REGION Network 3: Reset counter for write modbus parameter
   RUNG wire#powerrail
      { S7_Templates := "SrcType := Int" } GT_Contact(in1 := "PCS1".iCountDoneW, in2 := 9)
      Move(in := 1, out1 => "PCS1".iCountDoneW)
   END_RUNG
   // the same network as SCL:
   IF "PCS1".iCountDoneW > 9 THEN "PCS1".iCountDoneW := 1; END_IF;
END_REGION

REGION Network 4: Counter for read modbus data value
   RUNG wire#powerrail
      N_Contact(operand := "MbPCS1_W".DONE, bit := "xPEP2")
      { S7_Templates := "SrcType := Int" } Add(in1 := "PCS1".iCountReadW, in2 := 1, out => "PCS1".iCountReadW)
   END_RUNG
   // the same network as SCL:
   #_w1 := NOT "MbPCS1_W".DONE AND "xPEP2";   // falling edge of "MbPCS1_W".DONE
   "xPEP2" := "MbPCS1_W".DONE;
   IF #_w1 THEN "PCS1".iCountReadW := "PCS1".iCountReadW + 1; END_IF;
END_REGION

REGION Network 5: Reset counter for read modbus data value
   RUNG wire#powerrail
      { S7_Templates := "SrcType := Int" } GT_Contact(in1 := "PCS1".iCountReadW, in2 := 9)
      Move(in := 1, out1 => "PCS1".iCountReadW)
   END_RUNG
   // the same network as SCL:
   IF "PCS1".iCountReadW > 9 THEN "PCS1".iCountReadW := 1; END_IF;
END_REGION

REGION Network 6: Set request data modbus
   RUNG wire#powerrail
      N_Contact(operand := "MbPCS1_W".DONE, bit := "xPEP3")
      S_Coil( "PCS1".xREQW )
   END_RUNG
   // the same network as SCL:
   #_w1 := NOT "MbPCS1_W".DONE AND "xPEP3";   // falling edge of "MbPCS1_W".DONE
   "xPEP3" := "MbPCS1_W".DONE;
   IF #_w1 THEN "PCS1".xREQW := TRUE; END_IF;
END_REGION

REGION Network 7: Reset request data modbus
   RUNG wire#powerrail
      P_Contact(operand := "MbPCS1_W".DONE, bit := "xPEP4")
      R_Coil( "PCS1".xREQW )
   END_RUNG
   // the same network as SCL:
   #_w1 := "MbPCS1_W".DONE AND NOT "xPEP4";   // rising edge of "MbPCS1_W".DONE
   "xPEP4" := "MbPCS1_W".DONE;
   IF #_w1 THEN "PCS1".xREQW := FALSE; END_IF;
END_REGION

REGION Network 9: Write W_Block1 parameter
   // wUserPswIns
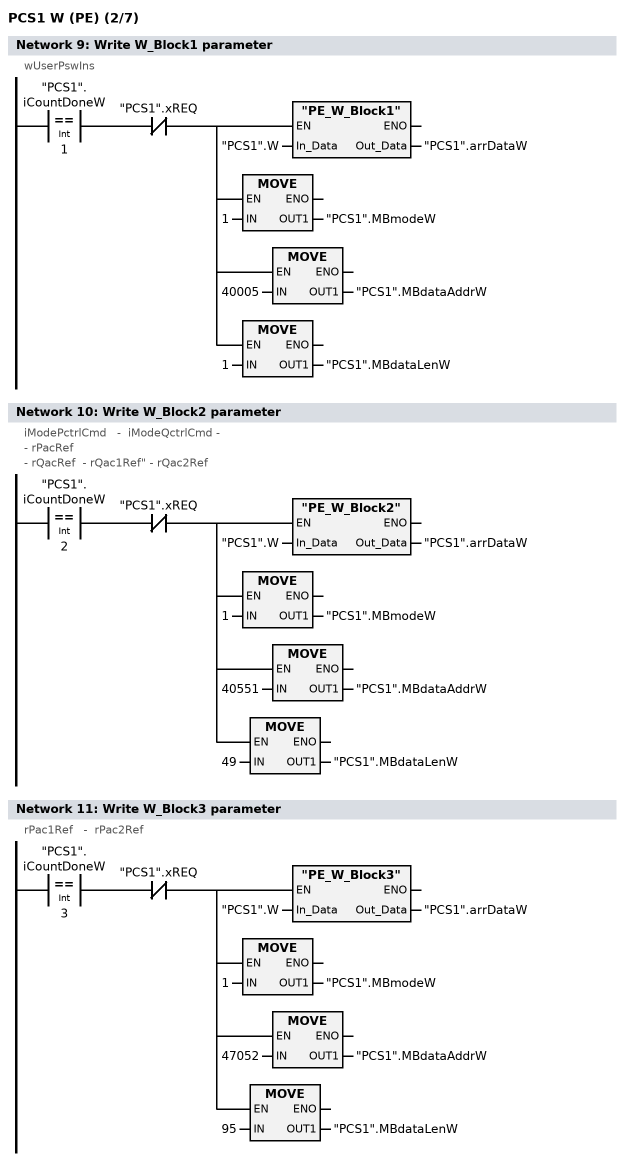
   RUNG wire#powerrail
      { S7_Templates := "SrcType := Int" } EQ_Contact(in1 := "PCS1".iCountDoneW, in2 := 1)
      I_Contact( "PCS1".xREQ )
      wire#w1
      "PE_W_Block1"(In_Data := "PCS1".W, Out_Data => "PCS1".arrDataW)
   END_RUNG
   RUNG wire#w1
      Move(in := 1, out1 => "PCS1".MBmodeW)
   END_RUNG
   RUNG wire#w1
      Move(in := 40005, out1 => "PCS1".MBdataAddrW)
   END_RUNG
   RUNG wire#w1
      Move(in := 1, out1 => "PCS1".MBdataLenW)
   END_RUNG
   // the same network as SCL:
   #_w1 := ("PCS1".iCountDoneW = 1) AND NOT "PCS1".xREQ;
   IF #_w1 THEN
       "PE_W_Block1"(In_Data := "PCS1".W, Out_Data => "PCS1".arrDataW);
       "PCS1".MBmodeW := 1;
       "PCS1".MBdataAddrW := 40005;
       "PCS1".MBdataLenW := 1;
   END_IF;
END_REGION

REGION Network 10: Write W_Block2 parameter
   // iModePctrlCmd   -  iModeQctrlCmd - 
   // - rPacRef 
   // - rQacRef  - rQac1Ref" - rQac2Ref
   RUNG wire#powerrail
      { S7_Templates := "SrcType := Int" } EQ_Contact(in1 := "PCS1".iCountDoneW, in2 := 2)
      I_Contact( "PCS1".xREQ )
      wire#w1
      "PE_W_Block2"(In_Data := "PCS1".W, Out_Data => "PCS1".arrDataW)
   END_RUNG
   RUNG wire#w1
      Move(in := 1, out1 => "PCS1".MBmodeW)
   END_RUNG
   RUNG wire#w1
      Move(in := 40551, out1 => "PCS1".MBdataAddrW)
   END_RUNG
   RUNG wire#w1
      Move(in := 49, out1 => "PCS1".MBdataLenW)
   END_RUNG
   // the same network as SCL:
   #_w1 := ("PCS1".iCountDoneW = 2) AND NOT "PCS1".xREQ;
   IF #_w1 THEN
       "PE_W_Block2"(In_Data := "PCS1".W, Out_Data => "PCS1".arrDataW);
       "PCS1".MBmodeW := 1;
       "PCS1".MBdataAddrW := 40551;
       "PCS1".MBdataLenW := 49;
   END_IF;
END_REGION

REGION Network 11: Write W_Block3 parameter
   // rPac1Ref   -  rPac2Ref
   RUNG wire#powerrail
      { S7_Templates := "SrcType := Int" } EQ_Contact(in1 := "PCS1".iCountDoneW, in2 := 3)
      I_Contact( "PCS1".xREQ )
      wire#w1
      "PE_W_Block3"(In_Data := "PCS1".W, Out_Data => "PCS1".arrDataW)
   END_RUNG
   RUNG wire#w1
      Move(in := 1, out1 => "PCS1".MBmodeW)
   END_RUNG
   RUNG wire#w1
      Move(in := 47052, out1 => "PCS1".MBdataAddrW)
   END_RUNG
   RUNG wire#w1
      Move(in := 95, out1 => "PCS1".MBdataLenW)
   END_RUNG
   // the same network as SCL:
   #_w1 := ("PCS1".iCountDoneW = 3) AND NOT "PCS1".xREQ;
   IF #_w1 THEN
       "PE_W_Block3"(In_Data := "PCS1".W, Out_Data => "PCS1".arrDataW);
       "PCS1".MBmodeW := 1;
       "PCS1".MBdataAddrW := 47052;
       "PCS1".MBdataLenW := 95;
   END_IF;
END_REGION

REGION Network 12: Write Command Start
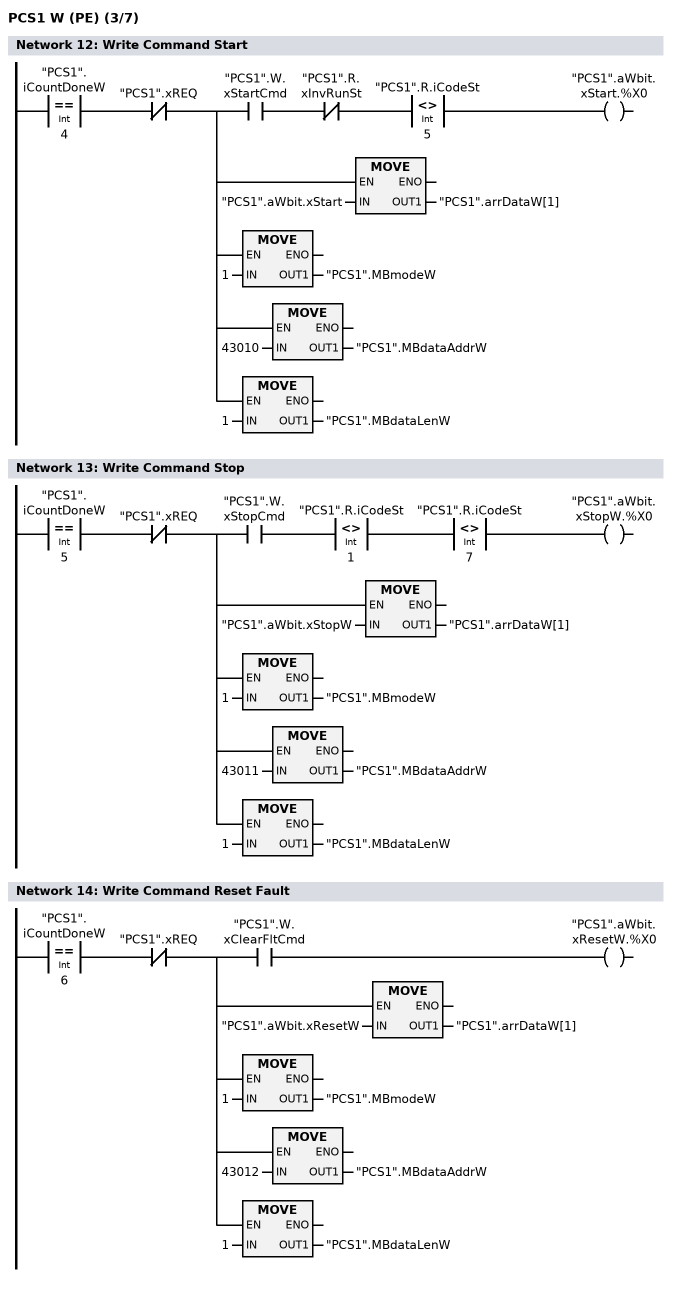
   RUNG wire#powerrail
      { S7_Templates := "SrcType := Int" } EQ_Contact(in1 := "PCS1".iCountDoneW, in2 := 4)
      I_Contact( "PCS1".xREQ )
      wire#w1
      Contact( "PCS1".W.xStartCmd )
      I_Contact( "PCS1".R.xInvRunSt )
      { S7_Templates := "SrcType := Int" } NE_Contact(in1 := "PCS1".R.iCodeSt, in2 := 5)
      Coil( "PCS1".aWbit.xStart.%X0 )
   END_RUNG
   RUNG wire#w1
      Move(in := "PCS1".aWbit.xStart, out1 => "PCS1".arrDataW[1])
   END_RUNG
   RUNG wire#w1
      Move(in := 1, out1 => "PCS1".MBmodeW)
   END_RUNG
   RUNG wire#w1
      Move(in := 43010, out1 => "PCS1".MBdataAddrW)
   END_RUNG
   RUNG wire#w1
      Move(in := 1, out1 => "PCS1".MBdataLenW)
   END_RUNG
   // the same network as SCL:
   #_w1 := ("PCS1".iCountDoneW = 4) AND NOT "PCS1".xREQ;
   "PCS1".aWbit.xStart.%X0 := #_w1 AND "PCS1".W.xStartCmd AND NOT "PCS1".R.xInvRunSt AND ("PCS1".R.iCodeSt <> 5);
   IF #_w1 THEN
       "PCS1".arrDataW[1] := "PCS1".aWbit.xStart;
       "PCS1".MBmodeW := 1;
       "PCS1".MBdataAddrW := 43010;
       "PCS1".MBdataLenW := 1;
   END_IF;
END_REGION

REGION Network 13: Write Command Stop
   RUNG wire#powerrail
      { S7_Templates := "SrcType := Int" } EQ_Contact(in1 := "PCS1".iCountDoneW, in2 := 5)
      I_Contact( "PCS1".xREQ )
      wire#w1
      Contact( "PCS1".W.xStopCmd )
      { S7_Templates := "SrcType := Int" } NE_Contact(in1 := "PCS1".R.iCodeSt, in2 := 1)
      { S7_Templates := "SrcType := Int" } NE_Contact(in1 := "PCS1".R.iCodeSt, in2 := 7)
      Coil( "PCS1".aWbit.xStopW.%X0 )
   END_RUNG
   RUNG wire#w1
      Move(in := "PCS1".aWbit.xStopW, out1 => "PCS1".arrDataW[1])
   END_RUNG
   RUNG wire#w1
      Move(in := 1, out1 => "PCS1".MBmodeW)
   END_RUNG
   RUNG wire#w1
      Move(in := 43011, out1 => "PCS1".MBdataAddrW)
   END_RUNG
   RUNG wire#w1
      Move(in := 1, out1 => "PCS1".MBdataLenW)
   END_RUNG
   // the same network as SCL:
   #_w1 := ("PCS1".iCountDoneW = 5) AND NOT "PCS1".xREQ;
   "PCS1".aWbit.xStopW.%X0 := #_w1 AND "PCS1".W.xStopCmd AND ("PCS1".R.iCodeSt <> 1) AND ("PCS1".R.iCodeSt <> 7);
   IF #_w1 THEN
       "PCS1".arrDataW[1] := "PCS1".aWbit.xStopW;
       "PCS1".MBmodeW := 1;
       "PCS1".MBdataAddrW := 43011;
       "PCS1".MBdataLenW := 1;
   END_IF;
END_REGION

REGION Network 14: Write Command Reset Fault
   RUNG wire#powerrail
      { S7_Templates := "SrcType := Int" } EQ_Contact(in1 := "PCS1".iCountDoneW, in2 := 6)
      I_Contact( "PCS1".xREQ )
      wire#w1
      Contact( "PCS1".W.xClearFltCmd )
      Coil( "PCS1".aWbit.xResetW.%X0 )
   END_RUNG
   RUNG wire#w1
      Move(in := "PCS1".aWbit.xResetW, out1 => "PCS1".arrDataW[1])
   END_RUNG
   RUNG wire#w1
      Move(in := 1, out1 => "PCS1".MBmodeW)
   END_RUNG
   RUNG wire#w1
      Move(in := 43012, out1 => "PCS1".MBdataAddrW)
   END_RUNG
   RUNG wire#w1
      Move(in := 1, out1 => "PCS1".MBdataLenW)
   END_RUNG
   // the same network as SCL:
   #_w1 := ("PCS1".iCountDoneW = 6) AND NOT "PCS1".xREQ;
   "PCS1".aWbit.xResetW.%X0 := #_w1 AND "PCS1".W.xClearFltCmd;
   IF #_w1 THEN
       "PCS1".arrDataW[1] := "PCS1".aWbit.xResetW;
       "PCS1".MBmodeW := 1;
       "PCS1".MBdataAddrW := 43012;
       "PCS1".MBdataLenW := 1;
   END_IF;
END_REGION

REGION Network 15: Write Command Enable Start/Stop
   // Con versione vecchia si usava solo questo registro per marcia ed arresto.
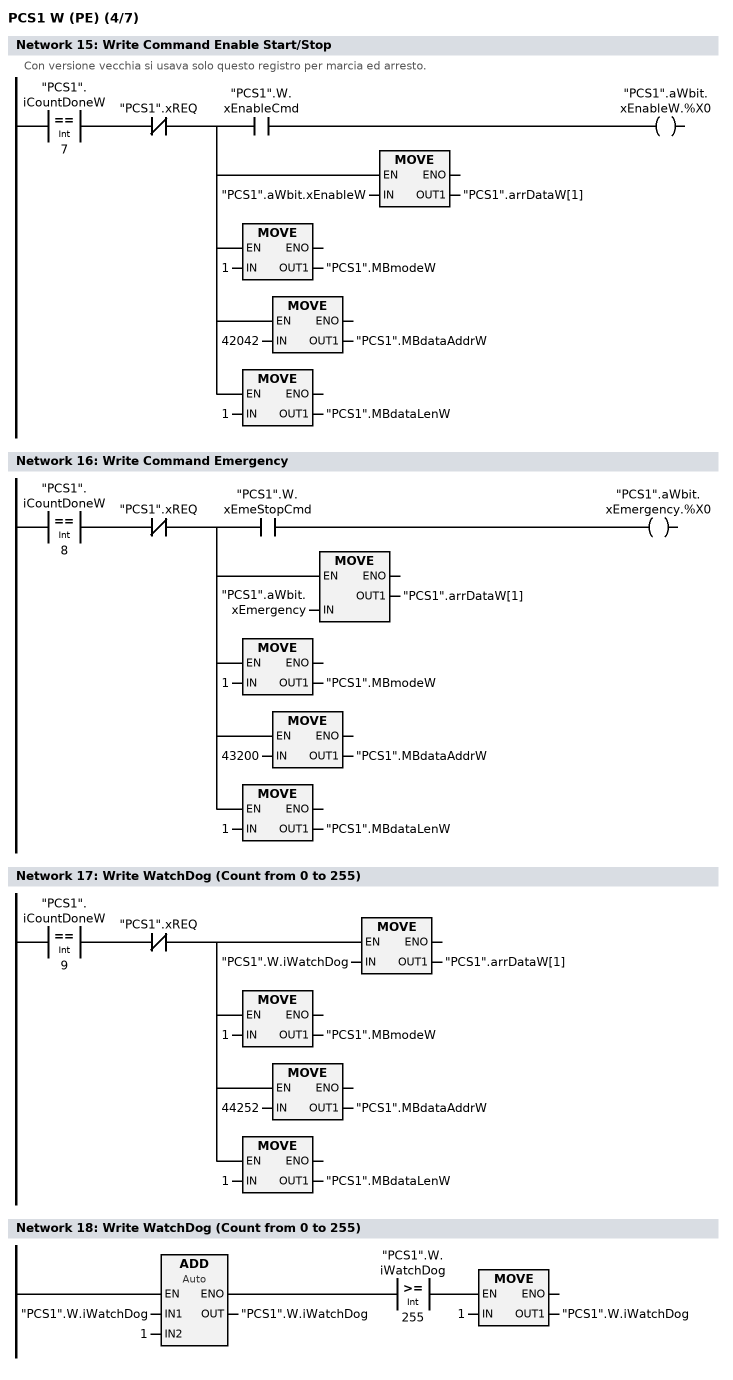
   RUNG wire#powerrail
      { S7_Templates := "SrcType := Int" } EQ_Contact(in1 := "PCS1".iCountDoneW, in2 := 7)
      I_Contact( "PCS1".xREQ )
      wire#w1
      Contact( "PCS1".W.xEnableCmd )
      Coil( "PCS1".aWbit.xEnableW.%X0 )
   END_RUNG
   RUNG wire#w1
      Move(in := "PCS1".aWbit.xEnableW, out1 => "PCS1".arrDataW[1])
   END_RUNG
   RUNG wire#w1
      Move(in := 1, out1 => "PCS1".MBmodeW)
   END_RUNG
   RUNG wire#w1
      Move(in := 42042, out1 => "PCS1".MBdataAddrW)
   END_RUNG
   RUNG wire#w1
      Move(in := 1, out1 => "PCS1".MBdataLenW)
   END_RUNG
   // the same network as SCL:
   #_w1 := ("PCS1".iCountDoneW = 7) AND NOT "PCS1".xREQ;
   "PCS1".aWbit.xEnableW.%X0 := #_w1 AND "PCS1".W.xEnableCmd;
   IF #_w1 THEN
       "PCS1".arrDataW[1] := "PCS1".aWbit.xEnableW;
       "PCS1".MBmodeW := 1;
       "PCS1".MBdataAddrW := 42042;
       "PCS1".MBdataLenW := 1;
   END_IF;
END_REGION

REGION Network 16: Write Command Emergency
   RUNG wire#powerrail
      { S7_Templates := "SrcType := Int" } EQ_Contact(in1 := "PCS1".iCountDoneW, in2 := 8)
      I_Contact( "PCS1".xREQ )
      wire#w1
      Contact( "PCS1".W.xEmeStopCmd )
      Coil( "PCS1".aWbit.xEmergency.%X0 )
   END_RUNG
   RUNG wire#w1
      Move(in := "PCS1".aWbit.xEmergency, out1 => "PCS1".arrDataW[1])
   END_RUNG
   RUNG wire#w1
      Move(in := 1, out1 => "PCS1".MBmodeW)
   END_RUNG
   RUNG wire#w1
      Move(in := 43200, out1 => "PCS1".MBdataAddrW)
   END_RUNG
   RUNG wire#w1
      Move(in := 1, out1 => "PCS1".MBdataLenW)
   END_RUNG
   // the same network as SCL:
   #_w1 := ("PCS1".iCountDoneW = 8) AND NOT "PCS1".xREQ;
   "PCS1".aWbit.xEmergency.%X0 := #_w1 AND "PCS1".W.xEmeStopCmd;
   IF #_w1 THEN
       "PCS1".arrDataW[1] := "PCS1".aWbit.xEmergency;
       "PCS1".MBmodeW := 1;
       "PCS1".MBdataAddrW := 43200;
       "PCS1".MBdataLenW := 1;
   END_IF;
END_REGION

REGION Network 17: Write WatchDog (Count from 0 to 255)
   RUNG wire#powerrail
      { S7_Templates := "SrcType := Int" } EQ_Contact(in1 := "PCS1".iCountDoneW, in2 := 9)
      I_Contact( "PCS1".xREQ )
      wire#w1
      Move(in := "PCS1".W.iWatchDog, out1 => "PCS1".arrDataW[1])
   END_RUNG
   RUNG wire#w1
      Move(in := 1, out1 => "PCS1".MBmodeW)
   END_RUNG
   RUNG wire#w1
      Move(in := 44252, out1 => "PCS1".MBdataAddrW)
   END_RUNG
   RUNG wire#w1
      Move(in := 1, out1 => "PCS1".MBdataLenW)
   END_RUNG
   // the same network as SCL:
   IF ("PCS1".iCountDoneW = 9) AND NOT "PCS1".xREQ THEN
       "PCS1".arrDataW[1] := "PCS1".W.iWatchDog;
       "PCS1".MBmodeW := 1;
       "PCS1".MBdataAddrW := 44252;
       "PCS1".MBdataLenW := 1;
   END_IF;
END_REGION

REGION Network 18: Write WatchDog (Count from 0 to 255)
   RUNG wire#powerrail
      Add(in1 := "PCS1".W.iWatchDog, in2 := 1, out => "PCS1".W.iWatchDog)
      { S7_Templates := "SrcType := Int" } GE_Contact(in1 := "PCS1".W.iWatchDog, in2 := 255)
      Move(in := 1, out1 => "PCS1".W.iWatchDog)
   END_RUNG
   // the same network as SCL:
   "PCS1".W.iWatchDog := "PCS1".W.iWatchDog + 1;
   IF "PCS1".W.iWatchDog >= 255 THEN "PCS1".W.iWatchDog := 1; END_IF;
END_REGION

REGION Network 20: 43010
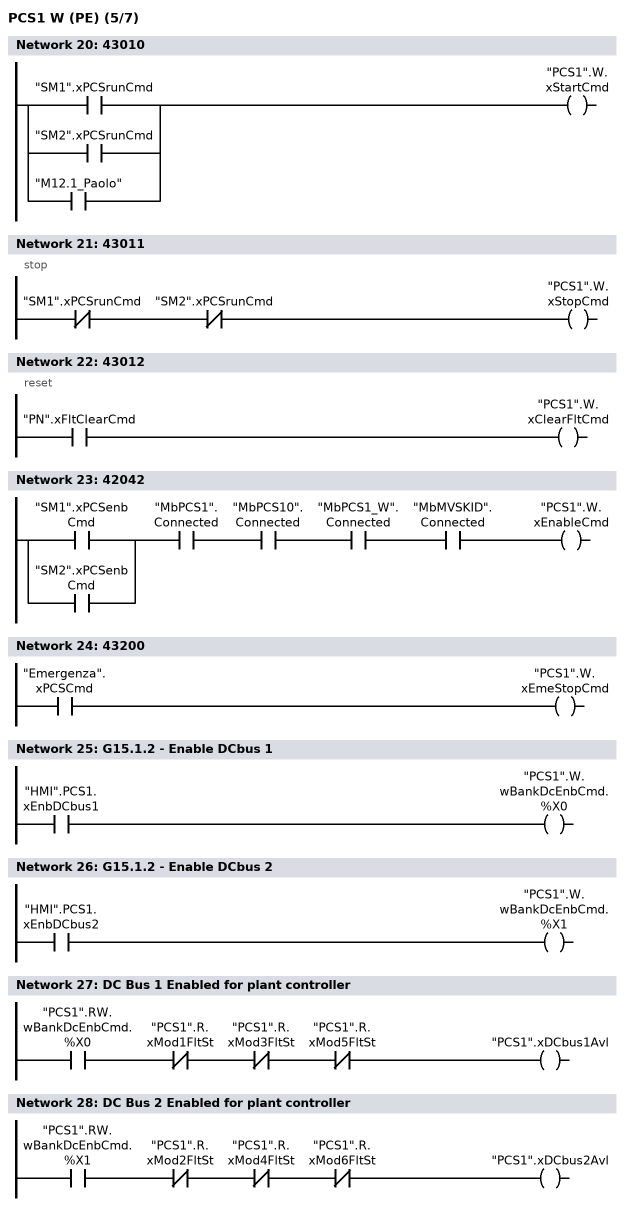
   RUNG wire#powerrail
      Contact( "SM1".xPCSrunCmd )
      wire#w1
      Coil( "PCS1".W.xStartCmd )
   END_RUNG
   RUNG wire#powerrail
      Contact( "SM2".xPCSrunCmd )
   END_RUNG wire#w1
   RUNG wire#powerrail
      Contact( "M12.1_Paolo" )
   END_RUNG wire#w1
   // the same network as SCL:
   "PCS1".W.xStartCmd := "SM1".xPCSrunCmd OR "SM2".xPCSrunCmd OR "M12.1_Paolo";
END_REGION

REGION Network 21: 43011
   // stop
   RUNG wire#powerrail
      I_Contact( "SM1".xPCSrunCmd )
      I_Contact( "SM2".xPCSrunCmd )
      Coil( "PCS1".W.xStopCmd )
   END_RUNG
   // the same network as SCL:
   "PCS1".W.xStopCmd := NOT "SM1".xPCSrunCmd AND NOT "SM2".xPCSrunCmd;
END_REGION

REGION Network 22: 43012
   // reset
   RUNG wire#powerrail
      Contact( "PN".xFltClearCmd )
      Coil( "PCS1".W.xClearFltCmd )
   END_RUNG
   // the same network as SCL:
   "PCS1".W.xClearFltCmd := "PN".xFltClearCmd;
END_REGION

REGION Network 23: 42042
   RUNG wire#powerrail
      Contact( "SM1".xPCSenbCmd )
      wire#w1
      Contact( "MbPCS1".Connected )
      Contact( "MbPCS10".Connected )
      Contact( "MbPCS1_W".Connected )
      Contact( "MbMVSKID".Connected )
      Coil( "PCS1".W.xEnableCmd )
   END_RUNG
   RUNG wire#powerrail
      Contact( "SM2".xPCSenbCmd )
   END_RUNG wire#w1
   // the same network as SCL:
   "PCS1".W.xEnableCmd := ("SM1".xPCSenbCmd OR "SM2".xPCSenbCmd) AND "MbPCS1".Connected AND "MbPCS10".Connected AND "MbPCS1_W".Connected AND "MbMVSKID".Connected;
END_REGION

REGION Network 24: 43200
   RUNG wire#powerrail
      Contact( "Emergenza".xPCSCmd )
      Coil( "PCS1".W.xEmeStopCmd )
   END_RUNG
   // the same network as SCL:
   "PCS1".W.xEmeStopCmd := "Emergenza".xPCSCmd;
END_REGION

REGION Network 25: G15.1.2 - Enable DCbus 1
   RUNG wire#powerrail
      Contact( "HMI".PCS1.xEnbDCbus1 )
      Coil( "PCS1".W.wBankDcEnbCmd.%X0 )
   END_RUNG
   // the same network as SCL:
   "PCS1".W.wBankDcEnbCmd.%X0 := "HMI".PCS1.xEnbDCbus1;
END_REGION

REGION Network 26: G15.1.2 - Enable DCbus 2
   RUNG wire#powerrail
      Contact( "HMI".PCS1.xEnbDCbus2 )
      Coil( "PCS1".W.wBankDcEnbCmd.%X1 )
   END_RUNG
   // the same network as SCL:
   "PCS1".W.wBankDcEnbCmd.%X1 := "HMI".PCS1.xEnbDCbus2;
END_REGION

REGION Network 27: DC Bus 1 Enabled for plant controller
   RUNG wire#powerrail
      Contact( "PCS1".RW.wBankDcEnbCmd.%X0 )
      I_Contact( "PCS1".R.xMod1FltSt )
      I_Contact( "PCS1".R.xMod3FltSt )
      I_Contact( "PCS1".R.xMod5FltSt )
      Coil( "PCS1".xDCbus1Avl )
   END_RUNG
   // the same network as SCL:
   "PCS1".xDCbus1Avl := "PCS1".RW.wBankDcEnbCmd.%X0 AND NOT "PCS1".R.xMod1FltSt AND NOT "PCS1".R.xMod3FltSt AND NOT "PCS1".R.xMod5FltSt;
END_REGION

REGION Network 28: DC Bus 2 Enabled for plant controller
   RUNG wire#powerrail
      Contact( "PCS1".RW.wBankDcEnbCmd.%X1 )
      I_Contact( "PCS1".R.xMod2FltSt )
      I_Contact( "PCS1".R.xMod4FltSt )
      I_Contact( "PCS1".R.xMod6FltSt )
      Coil( "PCS1".xDCbus2Avl )
   END_RUNG
   // the same network as SCL:
   "PCS1".xDCbus2Avl := "PCS1".RW.wBankDcEnbCmd.%X1 AND NOT "PCS1".R.xMod2FltSt AND NOT "PCS1".R.xMod4FltSt AND NOT "PCS1".R.xMod6FltSt;
END_REGION

REGION Network 30: Active Power local reference for PE with 2 DC Bus
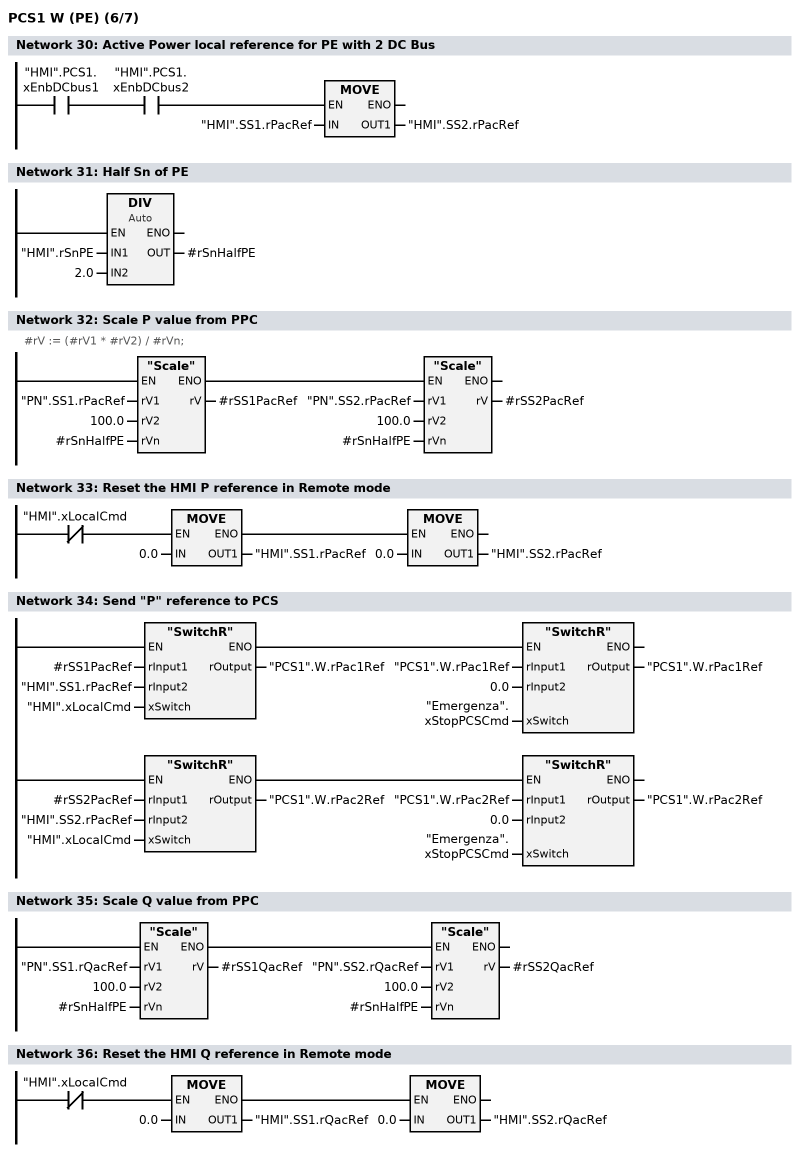
   RUNG wire#powerrail
      Contact( "HMI".PCS1.xEnbDCbus1 )
      Contact( "HMI".PCS1.xEnbDCbus2 )
      Move(in := "HMI".SS1.rPacRef, out1 => "HMI".SS2.rPacRef)
   END_RUNG
   // the same network as SCL:
   IF "HMI".PCS1.xEnbDCbus1 AND "HMI".PCS1.xEnbDCbus2 THEN "HMI".SS2.rPacRef := "HMI".SS1.rPacRef; END_IF;
END_REGION

REGION Network 31: Half Sn of PE
   RUNG wire#powerrail
      Div(in1 := "HMI".rSnPE, in2 := 2.0, out => #rSnHalfPE)
   END_RUNG
   // the same network as SCL:
   #rSnHalfPE := "HMI".rSnPE / 2.0;
END_REGION

REGION Network 32: Scale P value from PPC
   // #rV := (#rV1 * #rV2) / #rVn;
   RUNG wire#powerrail
      "Scale"(rV1 := "PN".SS1.rPacRef, rV2 := 100.0, rVn := #rSnHalfPE, rV => #rSS1PacRef)
      "Scale"(rV1 := "PN".SS2.rPacRef, rV2 := 100.0, rVn := #rSnHalfPE, rV => #rSS2PacRef)
   END_RUNG
   // the same network as SCL:
   "Scale"(rV1 := "PN".SS1.rPacRef, rV2 := 100.0, rVn := #rSnHalfPE, rV => #rSS1PacRef, ENO => #_w1);
   IF #_w1 THEN "Scale"(rV1 := "PN".SS2.rPacRef, rV2 := 100.0, rVn := #rSnHalfPE, rV => #rSS2PacRef); END_IF;
END_REGION

REGION Network 33: Reset the HMI P reference in Remote mode
   RUNG wire#powerrail
      I_Contact( "HMI".xLocalCmd )
      Move(in := 0.0, out1 => "HMI".SS1.rPacRef)
      Move(in := 0.0, out1 => "HMI".SS2.rPacRef)
   END_RUNG
   // the same network as SCL:
   IF NOT "HMI".xLocalCmd THEN
       "HMI".SS1.rPacRef := 0.0;
       "HMI".SS2.rPacRef := 0.0;
   END_IF;
END_REGION

REGION Network 34: Send "P" reference to PCS
   RUNG wire#powerrail
      "SwitchR"(rInput1 := #rSS1PacRef, rInput2 := "HMI".SS1.rPacRef, xSwitch := "HMI".xLocalCmd, rOutput => "PCS1".W.rPac1Ref)
      "SwitchR"(rInput1 := "PCS1".W.rPac1Ref, rInput2 := 0.0, xSwitch := "Emergenza".xStopPCSCmd, rOutput => "PCS1".W.rPac1Ref)
   END_RUNG
   RUNG wire#powerrail
      "SwitchR"(rInput1 := #rSS2PacRef, rInput2 := "HMI".SS2.rPacRef, xSwitch := "HMI".xLocalCmd, rOutput => "PCS1".W.rPac2Ref)
      "SwitchR"(rInput1 := "PCS1".W.rPac2Ref, rInput2 := 0.0, xSwitch := "Emergenza".xStopPCSCmd, rOutput => "PCS1".W.rPac2Ref)
   END_RUNG
   // the same network as SCL:
   "SwitchR"(rInput1 := #rSS1PacRef,
             rInput2 := "HMI".SS1.rPacRef,
             xSwitch := "HMI".xLocalCmd,
             rOutput => "PCS1".W.rPac1Ref,
             ENO => #_w1);
   IF #_w1 THEN
       "SwitchR"(rInput1 := "PCS1".W.rPac1Ref,
                 rInput2 := 0.0,
                 xSwitch := "Emergenza".xStopPCSCmd,
                 rOutput => "PCS1".W.rPac1Ref);
   END_IF;
   "SwitchR"(rInput1 := #rSS2PacRef,
             rInput2 := "HMI".SS2.rPacRef,
             xSwitch := "HMI".xLocalCmd,
             rOutput => "PCS1".W.rPac2Ref,
             ENO => #_w2);
   IF #_w2 THEN
       "SwitchR"(rInput1 := "PCS1".W.rPac2Ref,
                 rInput2 := 0.0,
                 xSwitch := "Emergenza".xStopPCSCmd,
                 rOutput => "PCS1".W.rPac2Ref);
   END_IF;
END_REGION

REGION Network 35: Scale Q value from PPC
   RUNG wire#powerrail
      "Scale"(rV1 := "PN".SS1.rQacRef, rV2 := 100.0, rVn := #rSnHalfPE, rV => #rSS1QacRef)
      "Scale"(rV1 := "PN".SS2.rQacRef, rV2 := 100.0, rVn := #rSnHalfPE, rV => #rSS2QacRef)
   END_RUNG
   // the same network as SCL:
   "Scale"(rV1 := "PN".SS1.rQacRef, rV2 := 100.0, rVn := #rSnHalfPE, rV => #rSS1QacRef, ENO => #_w1);
   IF #_w1 THEN "Scale"(rV1 := "PN".SS2.rQacRef, rV2 := 100.0, rVn := #rSnHalfPE, rV => #rSS2QacRef); END_IF;
END_REGION

REGION Network 36: Reset the HMI Q reference in Remote mode
   RUNG wire#powerrail
      I_Contact( "HMI".xLocalCmd )
      Move(in := 0.0, out1 => "HMI".SS1.rQacRef)
      Move(in := 0.0, out1 => "HMI".SS2.rQacRef)
   END_RUNG
   // the same network as SCL:
   IF NOT "HMI".xLocalCmd THEN
       "HMI".SS1.rQacRef := 0.0;
       "HMI".SS2.rQacRef := 0.0;
   END_IF;
END_REGION

REGION Network 37: Send "Q" reference to PCS
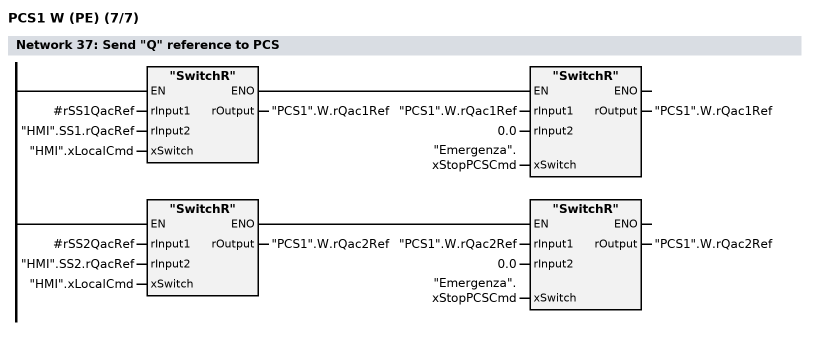
   RUNG wire#powerrail
      "SwitchR"(rInput1 := #rSS1QacRef, rInput2 := "HMI".SS1.rQacRef, xSwitch := "HMI".xLocalCmd, rOutput => "PCS1".W.rQac1Ref)
      "SwitchR"(rInput1 := "PCS1".W.rQac1Ref, rInput2 := 0.0, xSwitch := "Emergenza".xStopPCSCmd, rOutput => "PCS1".W.rQac1Ref)
   END_RUNG
   RUNG wire#powerrail
      "SwitchR"(rInput1 := #rSS2QacRef, rInput2 := "HMI".SS2.rQacRef, xSwitch := "HMI".xLocalCmd, rOutput => "PCS1".W.rQac2Ref)
      "SwitchR"(rInput1 := "PCS1".W.rQac2Ref, rInput2 := 0.0, xSwitch := "Emergenza".xStopPCSCmd, rOutput => "PCS1".W.rQac2Ref)
   END_RUNG
   // the same network as SCL:
   "SwitchR"(rInput1 := #rSS1QacRef,
             rInput2 := "HMI".SS1.rQacRef,
             xSwitch := "HMI".xLocalCmd,
             rOutput => "PCS1".W.rQac1Ref,
             ENO => #_w1);
   IF #_w1 THEN
       "SwitchR"(rInput1 := "PCS1".W.rQac1Ref,
                 rInput2 := 0.0,
                 xSwitch := "Emergenza".xStopPCSCmd,
                 rOutput => "PCS1".W.rQac1Ref);
   END_IF;
   "SwitchR"(rInput1 := #rSS2QacRef,
             rInput2 := "HMI".SS2.rQacRef,
             xSwitch := "HMI".xLocalCmd,
             rOutput => "PCS1".W.rQac2Ref,
             ENO => #_w2);
   IF #_w2 THEN
       "SwitchR"(rInput1 := "PCS1".W.rQac2Ref,
                 rInput2 := 0.0,
                 xSwitch := "Emergenza".xStopPCSCmd,
                 rOutput => "PCS1".W.rQac2Ref);
   END_IF;
END_REGION
END_FUNCTION

FUNCTION "PE_W_Block1" : Void
{ S7_Optimized_Access := 'TRUE' }
VERSION : 0.1
   VAR_INPUT 
      In_Data : "W_PE";   // pcs
   END_VAR

   VAR_OUTPUT 
      Out_Data : Array[1..125] of Word;
   END_VAR


BEGIN
	REGION
	    // 2022/01/24
	END_REGION
	
	REGION
	    
	    #Out_Data[1] := #In_Data."wUserPswIns";
	    
	END_REGION
END_FUNCTION

FUNCTION "PE_W_Block2" : Void
{ S7_Optimized_Access := 'TRUE' }
VERSION : 0.1
   VAR_INPUT 
      In_Data : "W_PE";   // udt. Samsung Data rack 1
   END_VAR

   VAR_OUTPUT 
      Out_Data : Array[1..125] of Word;
   END_VAR


BEGIN
	REGION
	    // 2022/01/24
	END_REGION
	
	REGION
	    
	    #Out_Data[1]    := INT_TO_WORD(#In_Data."iModePctrlCmd");
	    #Out_Data[2]    := INT_TO_WORD(#In_Data."iModeQctrlCmd");
	    #Out_Data[3]    := INT_TO_WORD(REAL_TO_INT((#In_Data."rPacRef")*100.0));
	    #Out_Data[8]    := INT_TO_WORD(REAL_TO_INT((#In_Data."rQacRef") * 100.0));
	    #Out_Data[48]   := INT_TO_WORD(REAL_TO_INT((#In_Data."rQac1Ref") * 100.0));
	    #Out_Data[49]   := INT_TO_WORD(REAL_TO_INT((#In_Data."rQac2Ref") * 100.0));
	    
	END_REGION
END_FUNCTION

FUNCTION "PE_W_Block3" : Void
{ S7_Optimized_Access := 'TRUE' }
VERSION : 0.1
   VAR_INPUT 
      In_Data : "W_PE";   // udt. Samsung Data rack 1
   END_VAR

   VAR_OUTPUT 
      Out_Data : Array[1..125] of Word;
   END_VAR


BEGIN
	REGION
	    // 2022/01/24
	END_REGION
	
	REGION
	    
	    #Out_Data[1]    := #In_Data."wBankDcEnbCmd";
	    #Out_Data[94]   := INT_TO_WORD(REAL_TO_INT((#In_Data."rPac1Ref")*100.0));
	    #Out_Data[95]   := INT_TO_WORD(REAL_TO_INT((#In_Data."rPac2Ref")*100.0));
	    
	END_REGION
END_FUNCTION

FUNCTION "Scale" : Void
{ S7_Optimized_Access := 'TRUE' }
VERSION : 0.1
   VAR_INPUT 
      rV1 : Real;
      rV2 : Real;
      rVn : Real;
   END_VAR

   VAR_OUTPUT 
      rV : Real;
   END_VAR


BEGIN
	
	#rV := (#rV1 * #rV2) / #rVn;
	
END_FUNCTION

FUNCTION "SwitchR" : Void
{ S7_Optimized_Access := 'TRUE' }
VERSION : 0.1
   VAR_INPUT 
      rInput1 : Real;
      rInput2 : Real;
      xSwitch : Bool;
   END_VAR

   VAR_OUTPUT 
      rOutput : Real;
   END_VAR

   VAR_TEMP 
      rOutTemp : Real;
   END_VAR


BEGIN
	IF #xSwitch THEN
	    #rOutTemp := #rInput2;
	ELSE
	    #rOutTemp := #rInput1;
	END_IF;
	
	#rOutput := #rOutTemp;
END_FUNCTION

FUNCTION "PN Com Read" : Void   // FC11, LAD
TITLE = ProfiNet Data Core <-> PEMS
{ S7_Optimized_Access := 'TRUE' }
VERSION : 0.1
// stored: AutoNumber false, IsIECCheckEnabled false, SetENOAutomatically false, UDAEnableTagReadback false
BEGIN

REGION Network 1: Read & Write Data From PEMS
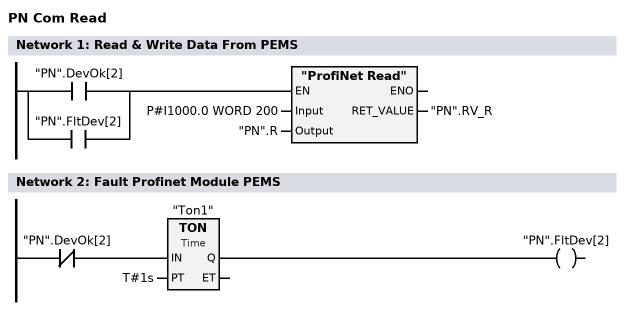
   RUNG wire#powerrail
      Contact( "PN".DevOk[2] )
      wire#w1
      "ProfiNet Read"(Input := P#I1000.0 WORD 200, Output := "PN".R, RET_VALUE => "PN".RV_R)
   END_RUNG
   RUNG wire#powerrail
      Contact( "PN".FltDev[2] )
   END_RUNG wire#w1
   // the same network as SCL:
   IF "PN".DevOk[2] OR "PN".FltDev[2] THEN
       "ProfiNet Read"(Input := P#I1000.0 WORD 200, Output := "PN".R, RET_VALUE => "PN".RV_R);
   END_IF;
END_REGION

REGION Network 2: Fault Profinet Module PEMS
   RUNG wire#powerrail
      I_Contact( "PN".DevOk[2] )
      { S7_Templates := "time_type := Time" } "Ton1".TON(pt := T#1s, et =>)
      Coil( "PN".FltDev[2] )
   END_RUNG
   // the same network as SCL:
   "Ton1".TON(IN := NOT "PN".DevOk[2], PT := T#1s);
   "PN".FltDev[2] := "Ton1".Q;
END_REGION
END_FUNCTION

FUNCTION "ProfiNet Read" : Void
{ S7_Optimized_Access := 'TRUE' }
VERSION : 0.1
   VAR_INPUT 
      Input : Variant;
   END_VAR

   VAR_OUTPUT 
      RET_VALUE : Int;
   END_VAR

   VAR_IN_OUT 
      Output : "PN Read";
   END_VAR

   VAR_TEMP 
      arrInput : Array[1..200] of Word;
      "DWORD" : DWord;
   END_VAR


BEGIN
	
	#RET_VALUE := MOVE_BLK_VARIANT(SRC := #Input, COUNT := 200, SRC_INDEX := 0, DEST_INDEX := 0, DEST => #arrInput);
	
	#Output."x1.1" := #arrInput[1].%X0;
	#Output."x1.2" := #arrInput[1].%X1;
	#Output."x1.3" := #arrInput[1].%X2;
	#Output."x1.4" := #arrInput[1].%X3;
	#Output."x1.5" := #arrInput[1].%X4;
	#Output."x1.6" := #arrInput[1].%X5;
	#Output."x1.7" := #arrInput[1].%X6;
	#Output."x1.8" := #arrInput[1].%X7;
	
	#Output."x2.1" := #arrInput[1].%X8;
	#Output."x2.2" := #arrInput[1].%X9;
	#Output."x2.3" := #arrInput[1].%X10;
	#Output."x2.4" := #arrInput[1].%X11;
	#Output."x2.5" := #arrInput[1].%X12;
	#Output."x2.6" := #arrInput[1].%X13;
	#Output."x2.7" := #arrInput[1].%X14;
	#Output."x2.8" := #arrInput[1].%X15;
	
	#Output."x3.1" := #arrInput[2].%X0;
	#Output."x3.2" := #arrInput[2].%X1;
	#Output."x3.3" := #arrInput[2].%X2;
	#Output."x3.4" := #arrInput[2].%X3;
	#Output."x3.5" := #arrInput[2].%X4;
	#Output."x3.6" := #arrInput[2].%X5;
	#Output."x3.7" := #arrInput[2].%X6;
	#Output."x3.8" := #arrInput[2].%X7;
	
	#Output."x4.1" := #arrInput[2].%X8;
	#Output."x4.2" := #arrInput[2].%X9;
	#Output."x4.3" := #arrInput[2].%X10;
	#Output."x4.4" := #arrInput[2].%X11;
	#Output."x4.5" := #arrInput[2].%X12;
	#Output."x4.6" := #arrInput[2].%X13;
	#Output."x4.7" := #arrInput[2].%X14;
	#Output."x4.8" := #arrInput[2].%X15;
	
	#Output."x5.1" := #arrInput[3].%X0;
	#Output."x5.2" := #arrInput[3].%X1;
	#Output."x5.3" := #arrInput[3].%X2;
	#Output."x5.4" := #arrInput[3].%X3;
	#Output."x5.5" := #arrInput[3].%X4;
	#Output."x5.6" := #arrInput[3].%X5;
	#Output."x5.7" := #arrInput[3].%X6;
	#Output."x5.8" := #arrInput[3].%X7;
	
	#Output."x6.1" := #arrInput[3].%X8;
	#Output."x6.2" := #arrInput[3].%X9;
	#Output."x6.3" := #arrInput[3].%X10;
	#Output."x6.4" := #arrInput[3].%X11;
	#Output."x6.5" := #arrInput[3].%X12;
	#Output."x6.6" := #arrInput[3].%X13;
	#Output."x6.7" := #arrInput[3].%X14;
	#Output."x6.8" := #arrInput[3].%X15;
	
	#Output."x7.1" := #arrInput[4].%X0;
	#Output."x7.2" := #arrInput[4].%X1;
	#Output."x7.3" := #arrInput[4].%X2;
	#Output."x7.4" := #arrInput[4].%X3;
	#Output."x7.5" := #arrInput[4].%X4;
	#Output."x7.6" := #arrInput[4].%X5;
	#Output."x7.7" := #arrInput[4].%X6;
	#Output."x7.8" := #arrInput[4].%X7;
	
	#Output."x8.1" := #arrInput[4].%X8;
	#Output."x8.2" := #arrInput[4].%X9;
	#Output."x8.3" := #arrInput[4].%X10;
	#Output."x8.4" := #arrInput[4].%X11;
	#Output."x8.5" := #arrInput[4].%X12;
	#Output."x8.6" := #arrInput[4].%X13;
	#Output."x8.7" := #arrInput[4].%X14;
	#Output."x8.8" := #arrInput[4].%X15;
	
	#Output."x9.1" := #arrInput[5].%X0;
	#Output."x9.2" := #arrInput[5].%X1;
	#Output."x9.3" := #arrInput[5].%X2;
	#Output."x9.4" := #arrInput[5].%X3;
	#Output."x9.5" := #arrInput[5].%X4;
	#Output."x9.6" := #arrInput[5].%X5;
	#Output."x9.7" := #arrInput[5].%X6;
	#Output."x9.8" := #arrInput[5].%X7;
	
	#Output."x10.1" := #arrInput[5].%X8;
	#Output."x10.2" := #arrInput[5].%X9;
	#Output."x10.3" := #arrInput[5].%X10;
	#Output."x10.4" := #arrInput[5].%X11;
	#Output."x10.5" := #arrInput[5].%X12;
	#Output."x10.6" := #arrInput[5].%X13;
	#Output."x10.7" := #arrInput[5].%X14;
	#Output."x10.8" := #arrInput[5].%X15;
	
	#Output.i1 := WORD_TO_INT(#arrInput[6]);
	#Output.i2 := WORD_TO_INT(#arrInput[7]);
	#Output.i3 := WORD_TO_INT(#arrInput[8]);
	#Output.i4 := WORD_TO_INT(#arrInput[9]);
	#Output.i5 := WORD_TO_INT(#arrInput[10]);
	#Output.i6 := WORD_TO_INT(#arrInput[11]);
	#Output.i7 := WORD_TO_INT(#arrInput[12]);
	#Output.i8 := WORD_TO_INT(#arrInput[13]);
	#Output.i9 := WORD_TO_INT(#arrInput[14]);
	#Output.i10 := WORD_TO_INT(#arrInput[15]);
	#Output.i11 := WORD_TO_INT(#arrInput[16]);
	#Output.i12 := WORD_TO_INT(#arrInput[17]);
	#Output.i13 := WORD_TO_INT(#arrInput[18]);
	#Output.i14 := WORD_TO_INT(#arrInput[19]);
	#Output.i15 := WORD_TO_INT(#arrInput[20]);
	#Output.i16 := WORD_TO_INT(#arrInput[21]);
	#Output.i17 := WORD_TO_INT(#arrInput[22]);
	#Output.i18 := WORD_TO_INT(#arrInput[23]);
	#Output.i19 := WORD_TO_INT(#arrInput[24]);
	#Output.i20 := WORD_TO_INT(#arrInput[25]);
	#Output.i21 := WORD_TO_INT(#arrInput[26]);
	#Output.i22 := WORD_TO_INT(#arrInput[27]);
	#Output.i23 := WORD_TO_INT(#arrInput[28]);
	#Output.i24 := WORD_TO_INT(#arrInput[29]);
	#Output.i25 := WORD_TO_INT(#arrInput[30]);
	#Output.i26 := WORD_TO_INT(#arrInput[31]);
	#Output.i27 := WORD_TO_INT(#arrInput[32]);
	#Output.i28 := WORD_TO_INT(#arrInput[33]);
	#Output.i29 := WORD_TO_INT(#arrInput[34]);
	#Output.i30 := WORD_TO_INT(#arrInput[35]);
	#Output.i31 := WORD_TO_INT(#arrInput[36]);
	#Output.i32 := WORD_TO_INT(#arrInput[37]);
	#Output.i33 := WORD_TO_INT(#arrInput[38]);
	#Output.i34 := WORD_TO_INT(#arrInput[39]);
	#Output.i35 := WORD_TO_INT(#arrInput[40]);
	
	#DWORD.%W0 := #arrInput[41];
	#DWORD.%W1 := #arrInput[42];
	#Output.r1 := DWORD_TO_REAL(#DWORD);
	#DWORD.%W0 := #arrInput[43];
	#DWORD.%W1 := #arrInput[44];
	#Output.r2 := DWORD_TO_REAL(#DWORD);
	#DWORD.%W0 := #arrInput[45];
	#DWORD.%W1 := #arrInput[46];
	#Output.r3 := DWORD_TO_REAL(#DWORD);
	#DWORD.%W0 := #arrInput[47];
	#DWORD.%W1 := #arrInput[48];
	#Output.r4 := DWORD_TO_REAL(#DWORD);
	#DWORD.%W0 := #arrInput[49];
	#DWORD.%W1 := #arrInput[50];
	#Output.r5 := DWORD_TO_REAL(#DWORD);
	#DWORD.%W0 := #arrInput[51];
	#DWORD.%W1 := #arrInput[52];
	#Output.r6 := DWORD_TO_REAL(#DWORD);
	#DWORD.%W0 := #arrInput[53];
	#DWORD.%W1 := #arrInput[54];
	#Output.r7 := DWORD_TO_REAL(#DWORD);
	#DWORD.%W0 := #arrInput[55];
	#DWORD.%W1 := #arrInput[56];
	#Output.r8 := DWORD_TO_REAL(#DWORD);
	#DWORD.%W0 := #arrInput[57];
	#DWORD.%W1 := #arrInput[58];
	#Output.r9 := DWORD_TO_REAL(#DWORD);
	#DWORD.%W0 := #arrInput[59];
	#DWORD.%W1 := #arrInput[60];
	#Output.r10 := DWORD_TO_REAL(#DWORD);
	#DWORD.%W0 := #arrInput[61];
	#DWORD.%W1 := #arrInput[62];
	#Output.r11 := DWORD_TO_REAL(#DWORD);
	#DWORD.%W0 := #arrInput[63];
	#DWORD.%W1 := #arrInput[64];
	#Output.r12 := DWORD_TO_REAL(#DWORD);
	#DWORD.%W0 := #arrInput[65];
	#DWORD.%W1 := #arrInput[66];
	#Output.r13 := DWORD_TO_REAL(#DWORD);
	#DWORD.%W0 := #arrInput[67];
	#DWORD.%W1 := #arrInput[68];
	#Output.r14 := DWORD_TO_REAL(#DWORD);
	#DWORD.%W0 := #arrInput[69];
	#DWORD.%W1 := #arrInput[70];
	#Output.r15 := DWORD_TO_REAL(#DWORD);
	#DWORD.%W0 := #arrInput[71];
	#DWORD.%W1 := #arrInput[72];
	#Output.r16 := DWORD_TO_REAL(#DWORD);
	#DWORD.%W0 := #arrInput[73];
	#DWORD.%W1 := #arrInput[74];
	#Output.r17 := DWORD_TO_REAL(#DWORD);
	#DWORD.%W0 := #arrInput[75];
	#DWORD.%W1 := #arrInput[76];
	#Output.r18 := DWORD_TO_REAL(#DWORD);
	#DWORD.%W0 := #arrInput[77];
	#DWORD.%W1 := #arrInput[78];
	#Output.r19 := DWORD_TO_REAL(#DWORD);
	#DWORD.%W0 := #arrInput[79];
	#DWORD.%W1 := #arrInput[80];
	#Output.r20 := DWORD_TO_REAL(#DWORD);
	#DWORD.%W0 := #arrInput[81];
	#DWORD.%W1 := #arrInput[82];
	#Output.r21 := DWORD_TO_REAL(#DWORD);
	#DWORD.%W0 := #arrInput[83];
	#DWORD.%W1 := #arrInput[84];
	#Output.r22 := DWORD_TO_REAL(#DWORD);
	#DWORD.%W0 := #arrInput[85];
	#DWORD.%W1 := #arrInput[86];
	#Output.r23 := DWORD_TO_REAL(#DWORD);
	#DWORD.%W0 := #arrInput[87];
	#DWORD.%W1 := #arrInput[88];
	#Output.r24 := DWORD_TO_REAL(#DWORD);
	#DWORD.%W0 := #arrInput[89];
	#DWORD.%W1 := #arrInput[90];
	#Output.r25 := DWORD_TO_REAL(#DWORD);
	#DWORD.%W0 := #arrInput[91];
	#DWORD.%W1 := #arrInput[92];
	#Output.r26 := DWORD_TO_REAL(#DWORD);
	#DWORD.%W0 := #arrInput[93];
	#DWORD.%W1 := #arrInput[94];
	#Output.r27 := DWORD_TO_REAL(#DWORD);
	#DWORD.%W0 := #arrInput[95];
	#DWORD.%W1 := #arrInput[96];
	#Output.r28 := DWORD_TO_REAL(#DWORD);
	#DWORD.%W0 := #arrInput[97];
	#DWORD.%W1 := #arrInput[98];
	#Output.r29 := DWORD_TO_REAL(#DWORD);
	#DWORD.%W0 := #arrInput[99];
	#DWORD.%W1 := #arrInput[100];
	#Output.r30 := DWORD_TO_REAL(#DWORD);
	#DWORD.%W0 := #arrInput[101];
	#DWORD.%W1 := #arrInput[102];
	#Output.r31 := DWORD_TO_REAL(#DWORD);
	#DWORD.%W0 := #arrInput[103];
	#DWORD.%W1 := #arrInput[104];
	#Output.r32 := DWORD_TO_REAL(#DWORD);
	#DWORD.%W0 := #arrInput[105];
	#DWORD.%W1 := #arrInput[106];
	#Output.r33 := DWORD_TO_REAL(#DWORD);
	#DWORD.%W0 := #arrInput[107];
	#DWORD.%W1 := #arrInput[108];
	#Output.r34 := DWORD_TO_REAL(#DWORD);
	#DWORD.%W0 := #arrInput[109];
	#DWORD.%W1 := #arrInput[110];
	#Output.r35 := DWORD_TO_REAL(#DWORD);
	#DWORD.%W0 := #arrInput[111];
	#DWORD.%W1 := #arrInput[112];
	#Output.r36 := DWORD_TO_REAL(#DWORD);
	#DWORD.%W0 := #arrInput[113];
	#DWORD.%W1 := #arrInput[114];
	#Output.r37 := DWORD_TO_REAL(#DWORD);
	#DWORD.%W0 := #arrInput[115];
	#DWORD.%W1 := #arrInput[116];
	#Output.r38 := DWORD_TO_REAL(#DWORD);
	#DWORD.%W0 := #arrInput[117];
	#DWORD.%W1 := #arrInput[118];
	#Output.r39 := DWORD_TO_REAL(#DWORD);
	#DWORD.%W0 := #arrInput[119];
	#DWORD.%W1 := #arrInput[120];
	#Output.r40 := DWORD_TO_REAL(#DWORD);
	#DWORD.%W0 := #arrInput[121];
	#DWORD.%W1 := #arrInput[122];
	#Output.r41 := DWORD_TO_REAL(#DWORD);
	#DWORD.%W0 := #arrInput[123];
	#DWORD.%W1 := #arrInput[124];
	#Output.r42 := DWORD_TO_REAL(#DWORD);
	#DWORD.%W0 := #arrInput[125];
	#DWORD.%W1 := #arrInput[126];
	#Output.r43 := DWORD_TO_REAL(#DWORD);
	#DWORD.%W0 := #arrInput[127];
	#DWORD.%W1 := #arrInput[128];
	#Output.r44 := DWORD_TO_REAL(#DWORD);
	#DWORD.%W0 := #arrInput[129];
	#DWORD.%W1 := #arrInput[130];
	#Output.r45 := DWORD_TO_REAL(#DWORD);
	#DWORD.%W0 := #arrInput[131];
	#DWORD.%W1 := #arrInput[132];
	#Output.r46 := DWORD_TO_REAL(#DWORD);
	#DWORD.%W0 := #arrInput[133];
	#DWORD.%W1 := #arrInput[134];
	#Output.r47 := DWORD_TO_REAL(#DWORD);
	#DWORD.%W0 := #arrInput[135];
	#DWORD.%W1 := #arrInput[136];
	#Output.r48 := DWORD_TO_REAL(#DWORD);
	#DWORD.%W0 := #arrInput[137];
	#DWORD.%W1 := #arrInput[138];
	#Output.r49 := DWORD_TO_REAL(#DWORD);
	#DWORD.%W0 := #arrInput[139];
	#DWORD.%W1 := #arrInput[140];
	#Output.r50 := DWORD_TO_REAL(#DWORD);
	#DWORD.%W0 := #arrInput[141];
	#DWORD.%W1 := #arrInput[142];
	#Output.r51 := DWORD_TO_REAL(#DWORD);
	#DWORD.%W0 := #arrInput[143];
	#DWORD.%W1 := #arrInput[144];
	#Output.r52 := DWORD_TO_REAL(#DWORD);
	#DWORD.%W0 := #arrInput[145];
	#DWORD.%W1 := #arrInput[146];
	#Output.r53 := DWORD_TO_REAL(#DWORD);
	#DWORD.%W0 := #arrInput[147];
	#DWORD.%W1 := #arrInput[148];
	#Output.r54 := DWORD_TO_REAL(#DWORD);
	#DWORD.%W0 := #arrInput[149];
	#DWORD.%W1 := #arrInput[150];
	#Output.r55 := DWORD_TO_REAL(#DWORD);
	#DWORD.%W0 := #arrInput[151];
	#DWORD.%W1 := #arrInput[152];
	#Output.r56 := DWORD_TO_REAL(#DWORD);
	#DWORD.%W0 := #arrInput[153];
	#DWORD.%W1 := #arrInput[154];
	#Output.r57 := DWORD_TO_REAL(#DWORD);
	#DWORD.%W0 := #arrInput[155];
	#DWORD.%W1 := #arrInput[156];
	#Output.r58 := DWORD_TO_REAL(#DWORD);
	#DWORD.%W0 := #arrInput[157];
	#DWORD.%W1 := #arrInput[158];
	#Output.r59 := DWORD_TO_REAL(#DWORD);
	#DWORD.%W0 := #arrInput[159];
	#DWORD.%W1 := #arrInput[160];
	#Output.r60 := DWORD_TO_REAL(#DWORD);
	#DWORD.%W0 := #arrInput[161];
	#DWORD.%W1 := #arrInput[162];
	#Output.r61 := DWORD_TO_REAL(#DWORD);
	#DWORD.%W0 := #arrInput[163];
	#DWORD.%W1 := #arrInput[164];
	#Output.r62 := DWORD_TO_REAL(#DWORD);
	#DWORD.%W0 := #arrInput[165];
	#DWORD.%W1 := #arrInput[166];
	#Output.r63 := DWORD_TO_REAL(#DWORD);
	#DWORD.%W0 := #arrInput[167];
	#DWORD.%W1 := #arrInput[168];
	#Output.r64 := DWORD_TO_REAL(#DWORD);
	#DWORD.%W0 := #arrInput[169];
	#DWORD.%W1 := #arrInput[170];
	#Output.r65 := DWORD_TO_REAL(#DWORD);
	#DWORD.%W0 := #arrInput[171];
	#DWORD.%W1 := #arrInput[172];
	#Output.r66 := DWORD_TO_REAL(#DWORD);
	#DWORD.%W0 := #arrInput[173];
	#DWORD.%W1 := #arrInput[174];
	#Output.r67 := DWORD_TO_REAL(#DWORD);
	#DWORD.%W0 := #arrInput[175];
	#DWORD.%W1 := #arrInput[176];
	#Output.r68 := DWORD_TO_REAL(#DWORD);
	#DWORD.%W0 := #arrInput[177];
	#DWORD.%W1 := #arrInput[178];
	#Output.r69 := DWORD_TO_REAL(#DWORD);
	#DWORD.%W0 := #arrInput[179];
	#DWORD.%W1 := #arrInput[180];
	#Output.r70 := DWORD_TO_REAL(#DWORD);
	#DWORD.%W0 := #arrInput[181];
	#DWORD.%W1 := #arrInput[182];
	#Output.r71 := DWORD_TO_REAL(#DWORD);
	#DWORD.%W0 := #arrInput[183];
	#DWORD.%W1 := #arrInput[184];
	#Output.r72 := DWORD_TO_REAL(#DWORD);
	#DWORD.%W0 := #arrInput[185];
	#DWORD.%W1 := #arrInput[186];
	#Output.r73 := DWORD_TO_REAL(#DWORD);
	#DWORD.%W0 := #arrInput[187];
	#DWORD.%W1 := #arrInput[188];
	#Output.r74 := DWORD_TO_REAL(#DWORD);
	#DWORD.%W0 := #arrInput[189];
	#DWORD.%W1 := #arrInput[190];
	#Output.r75 := DWORD_TO_REAL(#DWORD);
	#DWORD.%W0 := #arrInput[191];
	#DWORD.%W1 := #arrInput[192];
	#Output.r76 := DWORD_TO_REAL(#DWORD);
	#DWORD.%W0 := #arrInput[193];
	#DWORD.%W1 := #arrInput[194];
	#Output.r77 := DWORD_TO_REAL(#DWORD);
	#DWORD.%W0 := #arrInput[195];
	#DWORD.%W1 := #arrInput[196];
	#Output.r78 := DWORD_TO_REAL(#DWORD);
	#DWORD.%W0 := #arrInput[197];
	#DWORD.%W1 := #arrInput[198];
	#Output.r79 := DWORD_TO_REAL(#DWORD);
	#DWORD.%W0 := #arrInput[199];
	#DWORD.%W1 := #arrInput[200];
	#Output.r80 := DWORD_TO_REAL(#DWORD);
	
END_FUNCTION

FUNCTION "PN Com Write" : Void   // FC12, LAD
TITLE = ProfiNet Data Core <-> PEMS
{ S7_Optimized_Access := 'TRUE' }
VERSION : 0.1
// stored: AutoNumber false, IsIECCheckEnabled false, SetENOAutomatically false, UDAEnableTagReadback false
BEGIN

REGION Network 1: Read & Write Data From PEMS
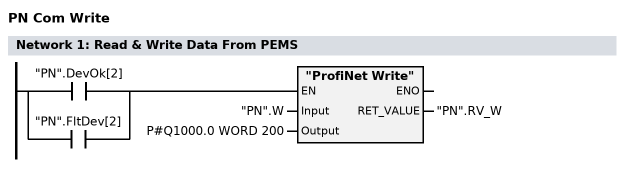
   RUNG wire#powerrail
      Contact( "PN".DevOk[2] )
      wire#w1
      "ProfiNet Write"(Input := "PN".W, Output := P#Q1000.0 WORD 200, RET_VALUE => "PN".RV_W)
   END_RUNG
   RUNG wire#powerrail
      Contact( "PN".FltDev[2] )
   END_RUNG wire#w1
   // the same network as SCL:
   IF "PN".DevOk[2] OR "PN".FltDev[2] THEN
       "ProfiNet Write"(Input := "PN".W, Output := P#Q1000.0 WORD 200, RET_VALUE => "PN".RV_W);
   END_IF;
END_REGION
END_FUNCTION

FUNCTION "ProfiNet Write" : Void
{ S7_Optimized_Access := 'TRUE' }
VERSION : 0.1
   VAR_INPUT 
      Input : "PN Write";
   END_VAR

   VAR_OUTPUT 
      RET_VALUE : Int;
   END_VAR

   VAR_IN_OUT 
      Output : Variant;
   END_VAR

   VAR_TEMP 
      arrOutput : Array[1..200] of Word;
      "DWORD" : DWord;
   END_VAR


BEGIN
	
	#arrOutput[1].%X0 := #Input."x1.1";
	#arrOutput[1].%X1 := #Input."x1.2";
	#arrOutput[1].%X2 := #Input."x1.3";
	#arrOutput[1].%X3 := #Input."x1.4";
	#arrOutput[1].%X4 := #Input."x1.5";
	#arrOutput[1].%X5 := #Input."x1.6";
	#arrOutput[1].%X6 := #Input."x1.7";
	#arrOutput[1].%X7 := #Input."x1.8";
	
	#arrOutput[1].%X8 := #Input."x2.1";
	#arrOutput[1].%X9 := #Input."x2.2";
	#arrOutput[1].%X10 := #Input."x2.3";
	#arrOutput[1].%X11 := #Input."x2.4";
	#arrOutput[1].%X12 := #Input."x2.5";
	#arrOutput[1].%X13 := #Input."x2.6";
	#arrOutput[1].%X14 := #Input."x2.7";
	#arrOutput[1].%X15 := #Input."x2.8";
	
	#arrOutput[2].%X0 := #Input."x3.1";
	#arrOutput[2].%X1 := #Input."x3.2";
	#arrOutput[2].%X2 := #Input."x3.3";
	#arrOutput[2].%X3 := #Input."x3.4";
	#arrOutput[2].%X4 := #Input."x3.5";
	#arrOutput[2].%X5 := #Input."x3.6";
	#arrOutput[2].%X6 := #Input."x3.7";
	#arrOutput[2].%X7 := #Input."x3.8";
	
	#arrOutput[2].%X8 := #Input."x4.1";
	#arrOutput[2].%X9 := #Input."x4.2";
	#arrOutput[2].%X10 := #Input."x4.3";
	#arrOutput[2].%X11 := #Input."x4.4";
	#arrOutput[2].%X12 := #Input."x4.5";
	#arrOutput[2].%X13 := #Input."x4.6";
	#arrOutput[2].%X14 := #Input."x4.7";
	#arrOutput[2].%X15 := #Input."x4.8";
	
	#arrOutput[3].%X0 := #Input."x5.1";
	#arrOutput[3].%X1 := #Input."x5.2";
	#arrOutput[3].%X2 := #Input."x5.3";
	#arrOutput[3].%X3 := #Input."x5.4";
	#arrOutput[3].%X4 := #Input."x5.5";
	#arrOutput[3].%X5 := #Input."x5.6";
	#arrOutput[3].%X6 := #Input."x5.7";
	#arrOutput[3].%X7 := #Input."x5.8";
	
	#arrOutput[3].%X8 := #Input."x6.1";
	#arrOutput[3].%X9 := #Input."x6.2";
	#arrOutput[3].%X10 := #Input."x6.3";
	#arrOutput[3].%X11 := #Input."x6.4";
	#arrOutput[3].%X12 := #Input."x6.5";
	#arrOutput[3].%X13 := #Input."x6.6";
	#arrOutput[3].%X14 := #Input."x6.7";
	#arrOutput[3].%X15 := #Input."x6.8";
	
	#arrOutput[4].%X0 := #Input."x7.1";
	#arrOutput[4].%X1 := #Input."x7.2";
	#arrOutput[4].%X2 := #Input."x7.3";
	#arrOutput[4].%X3 := #Input."x7.4";
	#arrOutput[4].%X4 := #Input."x7.5";
	#arrOutput[4].%X5 := #Input."x7.6";
	#arrOutput[4].%X6 := #Input."x7.7";
	#arrOutput[4].%X7 := #Input."x7.8";
	
	#arrOutput[4].%X8 := #Input."x8.1";
	#arrOutput[4].%X9 := #Input."x8.2";
	#arrOutput[4].%X10 := #Input."x8.3";
	#arrOutput[4].%X11 := #Input."x8.4";
	#arrOutput[4].%X12 := #Input."x8.5";
	#arrOutput[4].%X13 := #Input."x8.6";
	#arrOutput[4].%X14 := #Input."x8.7";
	#arrOutput[4].%X15 := #Input."x8.8";
	
	#arrOutput[5].%X0 := #Input."x9.1";
	#arrOutput[5].%X1 := #Input."x9.2";
	#arrOutput[5].%X2 := #Input."x9.3";
	#arrOutput[5].%X3 := #Input."x9.4";
	#arrOutput[5].%X4 := #Input."x9.5";
	#arrOutput[5].%X5 := #Input."x9.6";
	#arrOutput[5].%X6 := #Input."x9.7";
	#arrOutput[5].%X7 := #Input."x9.8";
	
	#arrOutput[5].%X8 := #Input."x10.1";
	#arrOutput[5].%X9 := #Input."x10.2";
	#arrOutput[5].%X10 := #Input."x10.3";
	#arrOutput[5].%X11 := #Input."x10.4";
	#arrOutput[5].%X12 := #Input."x10.5";
	#arrOutput[5].%X13 := #Input."x10.6";
	#arrOutput[5].%X14 := #Input."x10.7";
	#arrOutput[5].%X15 := #Input."x10.8";
	
	#arrOutput[6] := INT_TO_WORD(#Input.i1);
	#arrOutput[7] := INT_TO_WORD(#Input.i2);
	#arrOutput[8] := INT_TO_WORD(#Input.i3);
	#arrOutput[9] := INT_TO_WORD(#Input.i4);
	#arrOutput[10] := INT_TO_WORD(#Input.i5);
	#arrOutput[11] := INT_TO_WORD(#Input.i6);
	#arrOutput[12] := INT_TO_WORD(#Input.i7);
	#arrOutput[13] := INT_TO_WORD(#Input.i8);
	#arrOutput[14] := INT_TO_WORD(#Input.i9);
	#arrOutput[15] := INT_TO_WORD(#Input.i10);
	#arrOutput[16] := INT_TO_WORD(#Input.i11);
	#arrOutput[17] := INT_TO_WORD(#Input.i12);
	#arrOutput[18] := INT_TO_WORD(#Input.i13);
	#arrOutput[19] := INT_TO_WORD(#Input.i14);
	#arrOutput[20] := INT_TO_WORD(#Input.i15);
	#arrOutput[21] := INT_TO_WORD(#Input.i16);
	#arrOutput[22] := INT_TO_WORD(#Input.i17);
	#arrOutput[23] := INT_TO_WORD(#Input.i18);
	#arrOutput[24] := INT_TO_WORD(#Input.i19);
	#arrOutput[25] := INT_TO_WORD(#Input.i20);
	#arrOutput[26] := INT_TO_WORD(#Input.i21);
	#arrOutput[27] := INT_TO_WORD(#Input.i22);
	#arrOutput[28] := INT_TO_WORD(#Input.i23);
	#arrOutput[29] := INT_TO_WORD(#Input.i24);
	#arrOutput[30] := INT_TO_WORD(#Input.i25);
	#arrOutput[31] := INT_TO_WORD(#Input.i26);
	#arrOutput[32] := INT_TO_WORD(#Input.i27);
	#arrOutput[33] := INT_TO_WORD(#Input.i28);
	#arrOutput[34] := INT_TO_WORD(#Input.i29);
	#arrOutput[35] := INT_TO_WORD(#Input.i30);
	#arrOutput[36] := INT_TO_WORD(#Input.i31);
	#arrOutput[37] := INT_TO_WORD(#Input.i32);
	#arrOutput[38] := INT_TO_WORD(#Input.i33);
	#arrOutput[39] := INT_TO_WORD(#Input.i34);
	#arrOutput[40] := INT_TO_WORD(#Input.i35);
	
	#DWORD := REAL_TO_DWORD(#Input.r1);
	#arrOutput[41] := #DWORD.%W0;
	#arrOutput[42] := #DWORD.%W1;
	#DWORD := REAL_TO_DWORD(#Input.r2);
	#arrOutput[43] := #DWORD.%W0;
	#arrOutput[44] := #DWORD.%W1;
	#DWORD := REAL_TO_DWORD(#Input.r3);
	#arrOutput[45] := #DWORD.%W0;
	#arrOutput[46] := #DWORD.%W1;
	#DWORD := REAL_TO_DWORD(#Input.r4);
	#arrOutput[47] := #DWORD.%W0;
	#arrOutput[48] := #DWORD.%W1;
	#DWORD := REAL_TO_DWORD(#Input.r5);
	#arrOutput[49] := #DWORD.%W0;
	#arrOutput[50] := #DWORD.%W1;
	#DWORD := REAL_TO_DWORD(#Input.r6);
	#arrOutput[51] := #DWORD.%W0;
	#arrOutput[52] := #DWORD.%W1;
	#DWORD := REAL_TO_DWORD(#Input.r7);
	#arrOutput[53] := #DWORD.%W0;
	#arrOutput[54] := #DWORD.%W1;
	#DWORD := REAL_TO_DWORD(#Input.r8);
	#arrOutput[55] := #DWORD.%W0;
	#arrOutput[56] := #DWORD.%W1;
	#DWORD := REAL_TO_DWORD(#Input.r9);
	#arrOutput[57] := #DWORD.%W0;
	#arrOutput[58] := #DWORD.%W1;
	#DWORD := REAL_TO_DWORD(#Input.r10);
	#arrOutput[59] := #DWORD.%W0;
	#arrOutput[60] := #DWORD.%W1;
	#DWORD := REAL_TO_DWORD(#Input.r11);
	#arrOutput[61] := #DWORD.%W0;
	#arrOutput[62] := #DWORD.%W1;
	#DWORD := REAL_TO_DWORD(#Input.r12);
	#arrOutput[63] := #DWORD.%W0;
	#arrOutput[64] := #DWORD.%W1;
	#DWORD := REAL_TO_DWORD(#Input.r13);
	#arrOutput[65] := #DWORD.%W0;
	#arrOutput[66] := #DWORD.%W1;
	#DWORD := REAL_TO_DWORD(#Input.r14);
	#arrOutput[67] := #DWORD.%W0;
	#arrOutput[68] := #DWORD.%W1;
	#DWORD := REAL_TO_DWORD(#Input.r15);
	#arrOutput[69] := #DWORD.%W0;
	#arrOutput[70] := #DWORD.%W1;
	#DWORD := REAL_TO_DWORD(#Input.r16);
	#arrOutput[71] := #DWORD.%W0;
	#arrOutput[72] := #DWORD.%W1;
	#DWORD := REAL_TO_DWORD(#Input.r17);
	#arrOutput[73] := #DWORD.%W0;
	#arrOutput[74] := #DWORD.%W1;
	#DWORD := REAL_TO_DWORD(#Input.r18);
	#arrOutput[75] := #DWORD.%W0;
	#arrOutput[76] := #DWORD.%W1;
	#DWORD := REAL_TO_DWORD(#Input.r19);
	#arrOutput[77] := #DWORD.%W0;
	#arrOutput[78] := #DWORD.%W1;
	#DWORD := REAL_TO_DWORD(#Input.r20);
	#arrOutput[79] := #DWORD.%W0;
	#arrOutput[80] := #DWORD.%W1;
	#DWORD := REAL_TO_DWORD(#Input.r21);
	#arrOutput[81] := #DWORD.%W0;
	#arrOutput[82] := #DWORD.%W1;
	#DWORD := REAL_TO_DWORD(#Input.r22);
	#arrOutput[83] := #DWORD.%W0;
	#arrOutput[84] := #DWORD.%W1;
	#DWORD := REAL_TO_DWORD(#Input.r23);
	#arrOutput[85] := #DWORD.%W0;
	#arrOutput[86] := #DWORD.%W1;
	#DWORD := REAL_TO_DWORD(#Input.r24);
	#arrOutput[87] := #DWORD.%W0;
	#arrOutput[88] := #DWORD.%W1;
	#DWORD := REAL_TO_DWORD(#Input.r25);
	#arrOutput[89] := #DWORD.%W0;
	#arrOutput[90] := #DWORD.%W1;
	#DWORD := REAL_TO_DWORD(#Input.r26);
	#arrOutput[91] := #DWORD.%W0;
	#arrOutput[92] := #DWORD.%W1;
	#DWORD := REAL_TO_DWORD(#Input.r27);
	#arrOutput[93] := #DWORD.%W0;
	#arrOutput[94] := #DWORD.%W1;
	#DWORD := REAL_TO_DWORD(#Input.r28);
	#arrOutput[95] := #DWORD.%W0;
	#arrOutput[96] := #DWORD.%W1;
	#DWORD := REAL_TO_DWORD(#Input.r29);
	#arrOutput[97] := #DWORD.%W0;
	#arrOutput[98] := #DWORD.%W1;
	#DWORD := REAL_TO_DWORD(#Input.r30);
	#arrOutput[99] := #DWORD.%W0;
	#arrOutput[100] := #DWORD.%W1;
	#DWORD := REAL_TO_DWORD(#Input.r31);
	#arrOutput[101] := #DWORD.%W0;
	#arrOutput[102] := #DWORD.%W1;
	#DWORD := REAL_TO_DWORD(#Input.r32);
	#arrOutput[103] := #DWORD.%W0;
	#arrOutput[104] := #DWORD.%W1;
	#DWORD := REAL_TO_DWORD(#Input.r33);
	#arrOutput[105] := #DWORD.%W0;
	#arrOutput[106] := #DWORD.%W1;
	#DWORD := REAL_TO_DWORD(#Input.r34);
	#arrOutput[107] := #DWORD.%W0;
	#arrOutput[108] := #DWORD.%W1;
	#DWORD := REAL_TO_DWORD(#Input.r35);
	#arrOutput[109] := #DWORD.%W0;
	#arrOutput[110] := #DWORD.%W1;
	#DWORD := REAL_TO_DWORD(#Input.r36);
	#arrOutput[111] := #DWORD.%W0;
	#arrOutput[112] := #DWORD.%W1;
	#DWORD := REAL_TO_DWORD(#Input.r37);
	#arrOutput[113] := #DWORD.%W0;
	#arrOutput[114] := #DWORD.%W1;
	#DWORD := REAL_TO_DWORD(#Input.r38);
	#arrOutput[115] := #DWORD.%W0;
	#arrOutput[116] := #DWORD.%W1;
	#DWORD := REAL_TO_DWORD(#Input.r39);
	#arrOutput[117] := #DWORD.%W0;
	#arrOutput[118] := #DWORD.%W1;
	#DWORD := REAL_TO_DWORD(#Input.r40);
	#arrOutput[119] := #DWORD.%W0;
	#arrOutput[120] := #DWORD.%W1;
	#DWORD := REAL_TO_DWORD(#Input.r41);
	#arrOutput[121] := #DWORD.%W0;
	#arrOutput[122] := #DWORD.%W1;
	#DWORD := REAL_TO_DWORD(#Input.r42);
	#arrOutput[123] := #DWORD.%W0;
	#arrOutput[124] := #DWORD.%W1;
	#DWORD := REAL_TO_DWORD(#Input.r43);
	#arrOutput[125] := #DWORD.%W0;
	#arrOutput[126] := #DWORD.%W1;
	#DWORD := REAL_TO_DWORD(#Input.r44);
	#arrOutput[127] := #DWORD.%W0;
	#arrOutput[128] := #DWORD.%W1;
	#DWORD := REAL_TO_DWORD(#Input.r45);
	#arrOutput[129] := #DWORD.%W0;
	#arrOutput[130] := #DWORD.%W1;
	#DWORD := REAL_TO_DWORD(#Input.r46);
	#arrOutput[131] := #DWORD.%W0;
	#arrOutput[132] := #DWORD.%W1;
	#DWORD := REAL_TO_DWORD(#Input.r47);
	#arrOutput[133] := #DWORD.%W0;
	#arrOutput[134] := #DWORD.%W1;
	#DWORD := REAL_TO_DWORD(#Input.r48);
	#arrOutput[135] := #DWORD.%W0;
	#arrOutput[136] := #DWORD.%W1;
	#DWORD := REAL_TO_DWORD(#Input.r49);
	#arrOutput[137] := #DWORD.%W0;
	#arrOutput[138] := #DWORD.%W1;
	#DWORD := REAL_TO_DWORD(#Input.r50);
	#arrOutput[139] := #DWORD.%W0;
	#arrOutput[140] := #DWORD.%W1;
	#DWORD := REAL_TO_DWORD(#Input.r51);
	#arrOutput[141] := #DWORD.%W0;
	#arrOutput[142] := #DWORD.%W1;
	#DWORD := REAL_TO_DWORD(#Input.r52);
	#arrOutput[143] := #DWORD.%W0;
	#arrOutput[144] := #DWORD.%W1;
	#DWORD := REAL_TO_DWORD(#Input.r53);
	#arrOutput[145] := #DWORD.%W0;
	#arrOutput[146] := #DWORD.%W1;
	#DWORD := REAL_TO_DWORD(#Input.r54);
	#arrOutput[147] := #DWORD.%W0;
	#arrOutput[148] := #DWORD.%W1;
	#DWORD := REAL_TO_DWORD(#Input.r55);
	#arrOutput[149] := #DWORD.%W0;
	#arrOutput[150] := #DWORD.%W1;
	#DWORD := REAL_TO_DWORD(#Input.r56);
	#arrOutput[151] := #DWORD.%W0;
	#arrOutput[152] := #DWORD.%W1;
	#DWORD := REAL_TO_DWORD(#Input.r57);
	#arrOutput[153] := #DWORD.%W0;
	#arrOutput[154] := #DWORD.%W1;
	#DWORD := REAL_TO_DWORD(#Input.r58);
	#arrOutput[155] := #DWORD.%W0;
	#arrOutput[156] := #DWORD.%W1;
	#DWORD := REAL_TO_DWORD(#Input.r59);
	#arrOutput[157] := #DWORD.%W0;
	#arrOutput[158] := #DWORD.%W1;
	#DWORD := REAL_TO_DWORD(#Input.r60);
	#arrOutput[159] := #DWORD.%W0;
	#arrOutput[160] := #DWORD.%W1;
	#DWORD := REAL_TO_DWORD(#Input.r61);
	#arrOutput[161] := #DWORD.%W0;
	#arrOutput[162] := #DWORD.%W1;
	#DWORD := REAL_TO_DWORD(#Input.r62);
	#arrOutput[163] := #DWORD.%W0;
	#arrOutput[164] := #DWORD.%W1;
	#DWORD := REAL_TO_DWORD(#Input.r63);
	#arrOutput[165] := #DWORD.%W0;
	#arrOutput[166] := #DWORD.%W1;
	#DWORD := REAL_TO_DWORD(#Input.r64);
	#arrOutput[167] := #DWORD.%W0;
	#arrOutput[168] := #DWORD.%W1;
	#DWORD := REAL_TO_DWORD(#Input.r65);
	#arrOutput[169] := #DWORD.%W0;
	#arrOutput[170] := #DWORD.%W1;
	#DWORD := REAL_TO_DWORD(#Input.r66);
	#arrOutput[171] := #DWORD.%W0;
	#arrOutput[172] := #DWORD.%W1;
	#DWORD := REAL_TO_DWORD(#Input.r67);
	#arrOutput[173] := #DWORD.%W0;
	#arrOutput[174] := #DWORD.%W1;
	#DWORD := REAL_TO_DWORD(#Input.r68);
	#arrOutput[175] := #DWORD.%W0;
	#arrOutput[176] := #DWORD.%W1;
	#DWORD := REAL_TO_DWORD(#Input.r69);
	#arrOutput[177] := #DWORD.%W0;
	#arrOutput[178] := #DWORD.%W1;
	#DWORD := REAL_TO_DWORD(#Input.r70);
	#arrOutput[179] := #DWORD.%W0;
	#arrOutput[180] := #DWORD.%W1;
	#DWORD := REAL_TO_DWORD(#Input.r71);
	#arrOutput[181] := #DWORD.%W0;
	#arrOutput[182] := #DWORD.%W1;
	#DWORD := REAL_TO_DWORD(#Input.r72);
	#arrOutput[183] := #DWORD.%W0;
	#arrOutput[184] := #DWORD.%W1;
	#DWORD := REAL_TO_DWORD(#Input.r73);
	#arrOutput[185] := #DWORD.%W0;
	#arrOutput[186] := #DWORD.%W1;
	#DWORD := REAL_TO_DWORD(#Input.r74);
	#arrOutput[187] := #DWORD.%W0;
	#arrOutput[188] := #DWORD.%W1;
	#DWORD := REAL_TO_DWORD(#Input.r75);
	#arrOutput[189] := #DWORD.%W0;
	#arrOutput[190] := #DWORD.%W1;
	#DWORD := REAL_TO_DWORD(#Input.r76);
	#arrOutput[191] := #DWORD.%W0;
	#arrOutput[192] := #DWORD.%W1;
	#DWORD := REAL_TO_DWORD(#Input.r77);
	#arrOutput[193] := #DWORD.%W0;
	#arrOutput[194] := #DWORD.%W1;
	#DWORD := REAL_TO_DWORD(#Input.r78);
	#arrOutput[195] := #DWORD.%W0;
	#arrOutput[196] := #DWORD.%W1;
	#DWORD := REAL_TO_DWORD(#Input.r79);
	#arrOutput[197] := #DWORD.%W0;
	#arrOutput[198] := #DWORD.%W1;
	#DWORD := REAL_TO_DWORD(#Input.r80);
	#arrOutput[199] := #DWORD.%W0;
	#arrOutput[200] := #DWORD.%W1;
	
	#RET_VALUE := MOVE_BLK_VARIANT(SRC := #arrOutput, COUNT := 200, SRC_INDEX := 0, DEST_INDEX := 0, DEST => #Output);
	
END_FUNCTION

FUNCTION_BLOCK "Main_Safety_RTG1"   // FB501, F_LAD
{ S7_Optimized_Access := 'TRUE' }
VERSION : 0.1
// stored: AutoNumber false, IsIECCheckEnabled false, UDAEnableTagReadback false
BEGIN

REGION Network 1: Receive data from Core - new
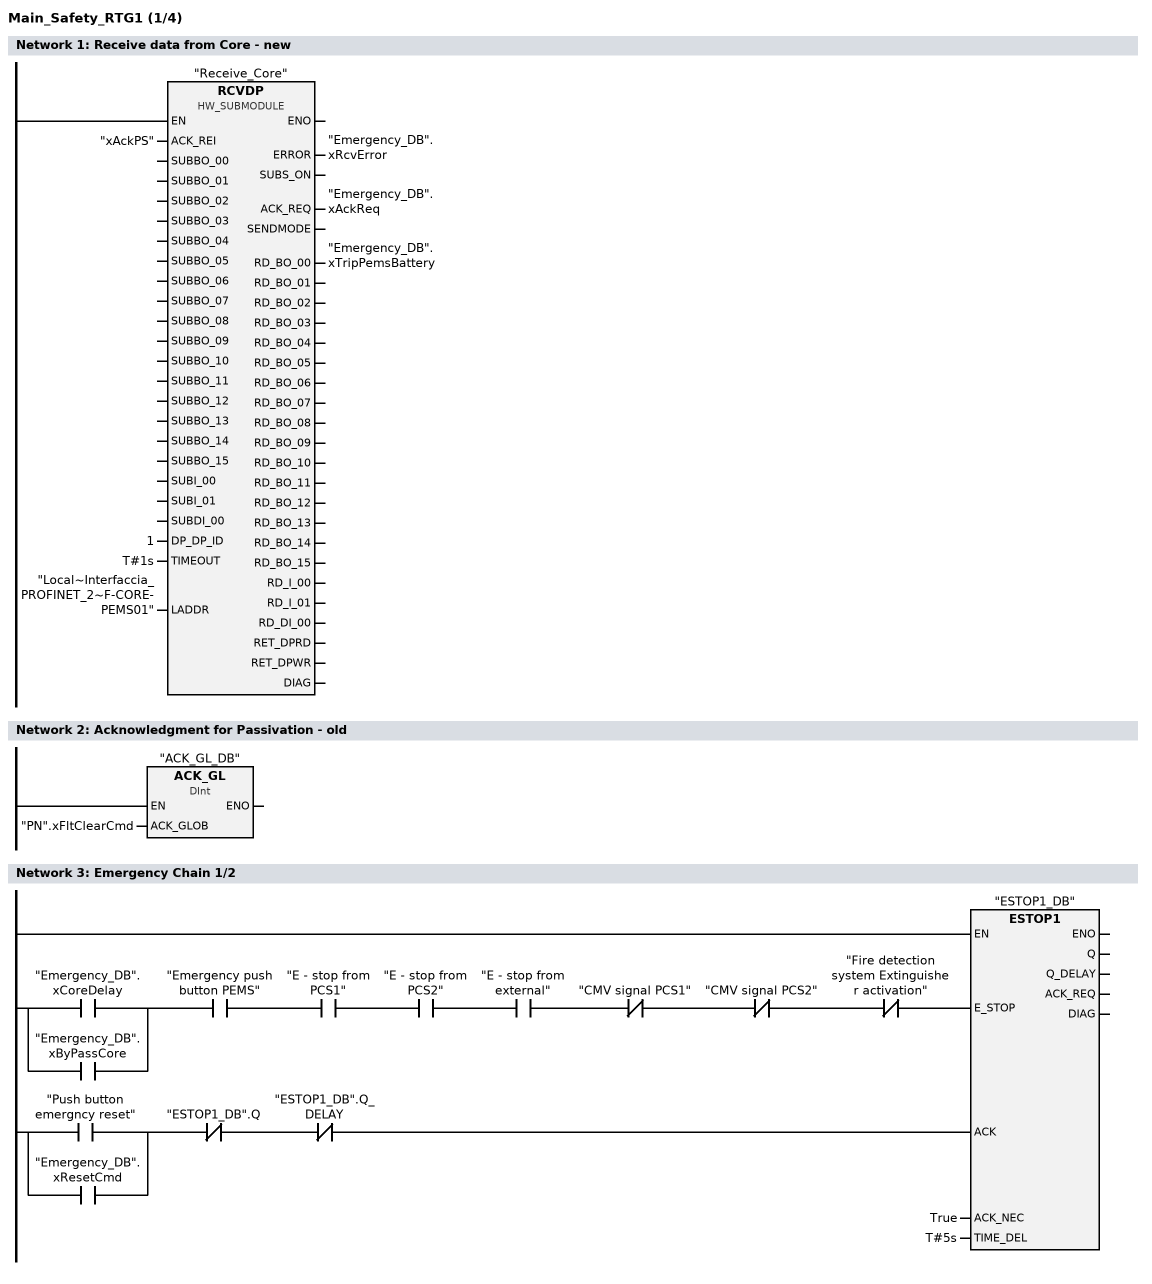
   RUNG wire#powerrail
      { S7_Templates := "laddr_type := HW_SUBMODULE" } "Receive_Core".RCVDP(ACK_REI := "xAckPS", SUBBO_00 :=, SUBBO_01 :=, SUBBO_02 :=, SUBBO_03 :=, SUBBO_04 :=, SUBBO_05 :=, SUBBO_06 :=, SUBBO_07 :=, SUBBO_08 :=, SUBBO_09 :=, SUBBO_10 :=, SUBBO_11 :=, SUBBO_12 :=, SUBBO_13 :=, SUBBO_14 :=, SUBBO_15 :=, SUBI_00 :=, SUBI_01 :=, SUBDI_00 :=, DP_DP_ID := 1, TIMEOUT := T#1s, LADDR := "Local~Interfaccia_PROFINET_2~F-CORE-PEMS01", ERROR => "Emergency_DB".xRcvError, SUBS_ON =>, ACK_REQ => "Emergency_DB".xAckReq, SENDMODE =>, RD_BO_00 => "Emergency_DB".xTripPemsBattery, RD_BO_01 =>, RD_BO_02 =>, RD_BO_03 =>, RD_BO_04 =>, RD_BO_05 =>, RD_BO_06 =>, RD_BO_07 =>, RD_BO_08 =>, RD_BO_09 =>, RD_BO_10 =>, RD_BO_11 =>, RD_BO_12 =>, RD_BO_13 =>, RD_BO_14 =>, RD_BO_15 =>, RD_I_00 =>, RD_I_01 =>, RD_DI_00 =>, RET_DPRD =>, RET_DPWR =>, DIAG =>)
   END_RUNG
   // the same network as SCL:
   "Receive_Core"(ACK_REI := "xAckPS",   // RCVDP
                  DP_DP_ID := 1,
                  TIMEOUT := T#1s,
                  LADDR := "Local~Interfaccia_PROFINET_2~F-CORE-PEMS01",
                  ERROR => "Emergency_DB".xRcvError,
                  ACK_REQ => "Emergency_DB".xAckReq,
                  RD_BO_00 => "Emergency_DB".xTripPemsBattery);
END_REGION

REGION Network 2: Acknowledgment for Passivation - old
   RUNG wire#powerrail
      { S7_Templates := "codedbool_type := DInt" } "ACK_GL_DB".ACK_GL(ACK_GLOB := "PN".xFltClearCmd)
   END_RUNG
   // the same network as SCL:
   "ACK_GL_DB"(ACK_GLOB := "PN".xFltClearCmd);   // ACK_GL
END_REGION

REGION Network 3: Emergency Chain 1/2
   RUNG wire#powerrail
      "ESTOP1_DB".ESTOP1(E_STOP := wire#w2, ACK := wire#w4, ACK_NEC := True, TIME_DEL := T#5s, Q =>, Q_DELAY =>, ACK_REQ =>, DIAG =>)
   END_RUNG
   RUNG wire#powerrail
      Contact( "Emergency_DB".xCoreDelay )
      wire#w1
      Contact( "Emergency push button PEMS" )
      Contact( "E - stop from PCS1" )
      Contact( "E - stop from PCS2" )
      Contact( "E - stop from external" )
      I_Contact( "CMV signal PCS1" )
      I_Contact( "CMV signal PCS2" )
      I_Contact( "Fire detection system Extinguisher activation" )
   END_RUNG wire#w2
   RUNG wire#powerrail
      Contact( "Emergency_DB".xByPassCore )
   END_RUNG wire#w1
   RUNG wire#powerrail
      Contact( "Push button emergncy reset" )
      wire#w3
      I_Contact( "ESTOP1_DB".Q )
      I_Contact( "ESTOP1_DB".Q_DELAY )
   END_RUNG wire#w4
   RUNG wire#powerrail
      Contact( "Emergency_DB".xResetCmd )
   END_RUNG wire#w3
   // the same network as SCL:
   "ESTOP1_DB"(E_STOP := ("Emergency_DB".xCoreDelay OR "Emergency_DB".xByPassCore) AND "Emergency push button PEMS" AND "E - stop from PCS1" AND "E - stop from PCS2" AND "E - stop from external" AND NOT "CMV signal PCS1" AND NOT "CMV signal PCS2" AND NOT "Fire detection system Extinguisher activation",   // ESTOP1
               ACK := ("Push button emergncy reset" OR "Emergency_DB".xResetCmd) AND NOT "ESTOP1_DB".Q AND NOT "ESTOP1_DB".Q_DELAY,
               ACK_NEC := True,
               TIME_DEL := T#5s);
END_REGION

REGION Network 4: Emergency shunt opening release RESET
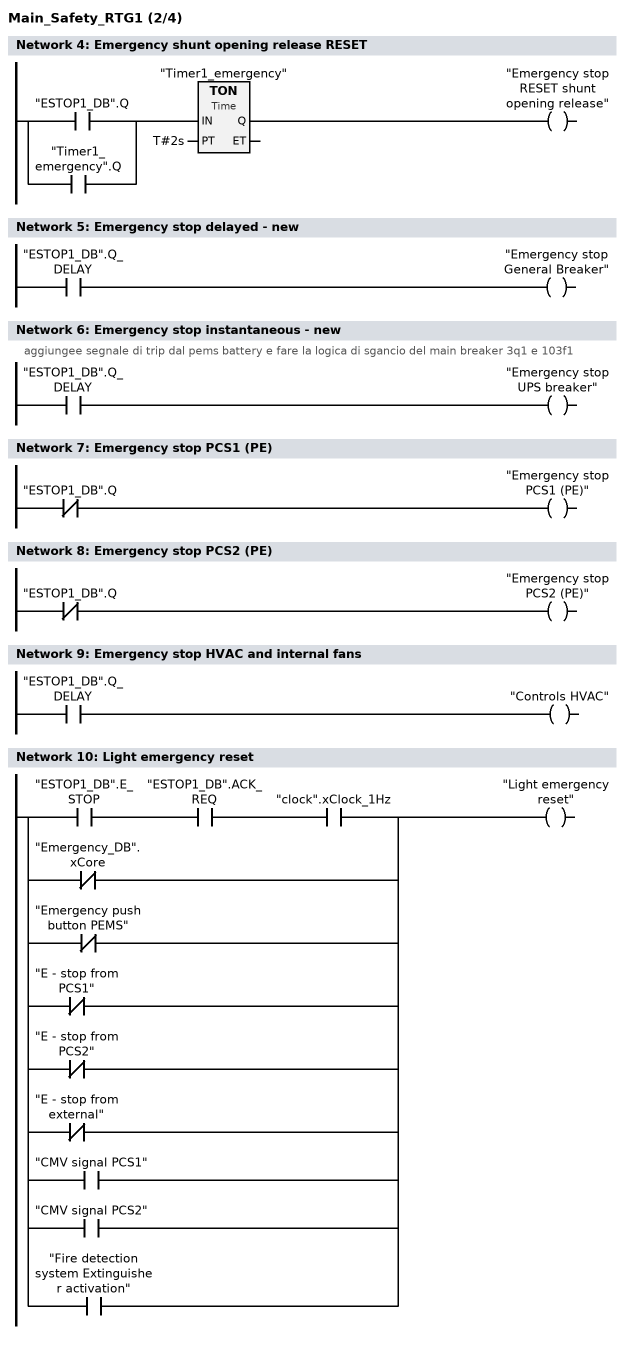
   RUNG wire#powerrail
      Contact( "ESTOP1_DB".Q )
      wire#w1
      { S7_Templates := "[time_type := Time, codedbool_type := DInt]" } "Timer1_emergency".TON(pt := T#2s, et =>)
      Coil( "Emergency stop RESET shunt opening release" )
   END_RUNG
   RUNG wire#powerrail
      Contact( "Timer1_emergency".Q )
   END_RUNG wire#w1
   // the same network as SCL:
   "Timer1_emergency".TON(IN := "ESTOP1_DB".Q OR "Timer1_emergency".Q, PT := T#2s);
   "Emergency stop RESET shunt opening release" := "Timer1_emergency".Q;
END_REGION

REGION Network 5: Emergency stop delayed - new
   RUNG wire#powerrail
      Contact( "ESTOP1_DB".Q_DELAY )
      Coil( "Emergency stop General Breaker" )
   END_RUNG
   // the same network as SCL:
   "Emergency stop General Breaker" := "ESTOP1_DB".Q_DELAY;
END_REGION

REGION Network 6: Emergency stop instantaneous - new
   // aggiungee segnale di trip dal pems battery e fare la logica di sgancio del main breaker 3q1 e 103f1
   RUNG wire#powerrail
      Contact( "ESTOP1_DB".Q_DELAY )
      Coil( "Emergency stop UPS breaker" )
   END_RUNG
   // the same network as SCL:
   "Emergency stop UPS breaker" := "ESTOP1_DB".Q_DELAY;
END_REGION

REGION Network 7: Emergency stop PCS1 (PE)
   RUNG wire#powerrail
      I_Contact( "ESTOP1_DB".Q )
      Coil( "Emergency stop PCS1 (PE)" )
   END_RUNG
   // the same network as SCL:
   "Emergency stop PCS1 (PE)" := NOT "ESTOP1_DB".Q;
END_REGION

REGION Network 8: Emergency stop PCS2 (PE)
   RUNG wire#powerrail
      I_Contact( "ESTOP1_DB".Q )
      Coil( "Emergency stop PCS2 (PE)" )
   END_RUNG
   // the same network as SCL:
   "Emergency stop PCS2 (PE)" := NOT "ESTOP1_DB".Q;
END_REGION

REGION Network 9: Emergency stop HVAC and internal fans
   RUNG wire#powerrail
      Contact( "ESTOP1_DB".Q_DELAY )
      Coil( "Controls HVAC" )
   END_RUNG
   // the same network as SCL:
   "Controls HVAC" := "ESTOP1_DB".Q_DELAY;
END_REGION

REGION Network 10: Light emergency reset
   RUNG wire#powerrail
      Contact( "ESTOP1_DB".E_STOP )
      Contact( "ESTOP1_DB".ACK_REQ )
      Contact( "clock".xClock_1Hz )
      wire#w1
      Coil( "Light emergency reset" )
   END_RUNG
   RUNG wire#powerrail
      I_Contact( "Emergency_DB".xCore )
   END_RUNG wire#w1
   RUNG wire#powerrail
      I_Contact( "Emergency push button PEMS" )
   END_RUNG wire#w1
   RUNG wire#powerrail
      I_Contact( "E - stop from PCS1" )
   END_RUNG wire#w1
   RUNG wire#powerrail
      I_Contact( "E - stop from PCS2" )
   END_RUNG wire#w1
   RUNG wire#powerrail
      I_Contact( "E - stop from external" )
   END_RUNG wire#w1
   RUNG wire#powerrail
      Contact( "CMV signal PCS1" )
   END_RUNG wire#w1
   RUNG wire#powerrail
      Contact( "CMV signal PCS2" )
   END_RUNG wire#w1
   RUNG wire#powerrail
      Contact( "Fire detection system Extinguisher activation" )
   END_RUNG wire#w1
   // the same network as SCL:
   "Light emergency reset" := ("ESTOP1_DB".E_STOP AND "ESTOP1_DB".ACK_REQ AND "clock".xClock_1Hz) OR NOT "Emergency_DB".xCore OR NOT "Emergency push button PEMS" OR NOT "E - stop from PCS1" OR NOT "E - stop from PCS2" OR NOT "E - stop from external" OR "CMV signal PCS1" OR "CMV signal PCS2" OR "Fire detection system Extinguisher activation";
END_REGION

REGION Network 11: Emergency - Open Battery Command
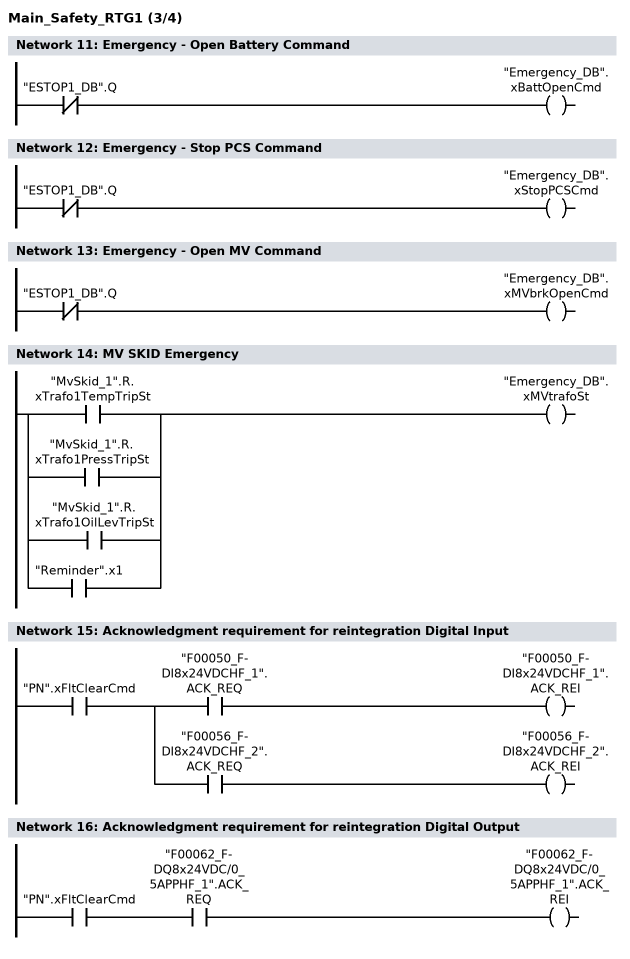
   RUNG wire#powerrail
      I_Contact( "ESTOP1_DB".Q )
      Coil( "Emergency_DB".xBattOpenCmd )
   END_RUNG
   // the same network as SCL:
   "Emergency_DB".xBattOpenCmd := NOT "ESTOP1_DB".Q;
END_REGION

REGION Network 12: Emergency - Stop PCS Command
   RUNG wire#powerrail
      I_Contact( "ESTOP1_DB".Q )
      Coil( "Emergency_DB".xStopPCSCmd )
   END_RUNG
   // the same network as SCL:
   "Emergency_DB".xStopPCSCmd := NOT "ESTOP1_DB".Q;
END_REGION

REGION Network 13: Emergency - Open MV Command
   RUNG wire#powerrail
      I_Contact( "ESTOP1_DB".Q )
      Coil( "Emergency_DB".xMVbrkOpenCmd )
   END_RUNG
   // the same network as SCL:
   "Emergency_DB".xMVbrkOpenCmd := NOT "ESTOP1_DB".Q;
END_REGION

REGION Network 14: MV SKID Emergency
   RUNG wire#powerrail
      Contact( "MvSkid_1".R.xTrafo1TempTripSt )
      wire#w1
      Coil( "Emergency_DB".xMVtrafoSt )
   END_RUNG
   RUNG wire#powerrail
      Contact( "MvSkid_1".R.xTrafo1PressTripSt )
   END_RUNG wire#w1
   RUNG wire#powerrail
      Contact( "MvSkid_1".R.xTrafo1OilLevTripSt )
   END_RUNG wire#w1
   RUNG wire#powerrail
      Contact( "Reminder".x1 )
   END_RUNG wire#w1
   // the same network as SCL:
   "Emergency_DB".xMVtrafoSt := "MvSkid_1".R.xTrafo1TempTripSt OR "MvSkid_1".R.xTrafo1PressTripSt OR "MvSkid_1".R.xTrafo1OilLevTripSt OR "Reminder".x1;
END_REGION

REGION Network 15: Acknowledgment requirement for reintegration Digital Input
   RUNG wire#powerrail
      Contact( "PN".xFltClearCmd )
      wire#w1
      Contact( "F00050_F-DI8x24VDCHF_1".ACK_REQ )
      Coil( "F00050_F-DI8x24VDCHF_1".ACK_REI )
   END_RUNG
   RUNG wire#w1
      Contact( "F00056_F-DI8x24VDCHF_2".ACK_REQ )
      Coil( "F00056_F-DI8x24VDCHF_2".ACK_REI )
   END_RUNG
   // the same network as SCL:
   "F00050_F-DI8x24VDCHF_1".ACK_REI := "PN".xFltClearCmd AND "F00050_F-DI8x24VDCHF_1".ACK_REQ;
   "F00056_F-DI8x24VDCHF_2".ACK_REI := "PN".xFltClearCmd AND "F00056_F-DI8x24VDCHF_2".ACK_REQ;
END_REGION

REGION Network 16: Acknowledgment requirement for reintegration Digital Output
   RUNG wire#powerrail
      Contact( "PN".xFltClearCmd )
      Contact( "F00062_F-DQ8x24VDC/0_5APPHF_1".ACK_REQ )
      Coil( "F00062_F-DQ8x24VDC/0_5APPHF_1".ACK_REI )
   END_RUNG
   // the same network as SCL:
   "F00062_F-DQ8x24VDC/0_5APPHF_1".ACK_REI := "PN".xFltClearCmd AND "F00062_F-DQ8x24VDC/0_5APPHF_1".ACK_REQ;
END_REGION

REGION Network 18: Send data to Core
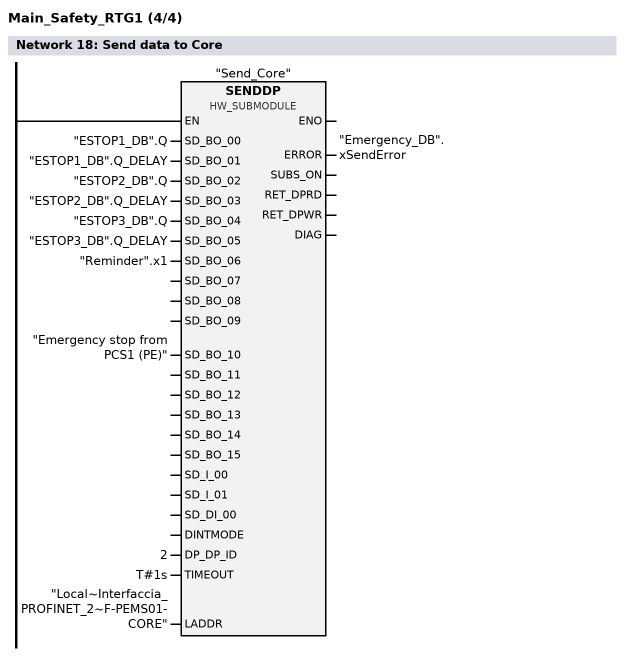
   RUNG wire#powerrail
      { S7_Templates := "laddr_type := HW_SUBMODULE" } "Send_Core".SENDDP(SD_BO_00 := "ESTOP1_DB".Q, SD_BO_01 := "ESTOP1_DB".Q_DELAY, SD_BO_02 := "ESTOP2_DB".Q, SD_BO_03 := "ESTOP2_DB".Q_DELAY, SD_BO_04 := "ESTOP3_DB".Q, SD_BO_05 := "ESTOP3_DB".Q_DELAY, SD_BO_06 := "Reminder".x1, SD_BO_07 :=, SD_BO_08 :=, SD_BO_09 :=, SD_BO_10 := "Emergency stop from PCS1 (PE)", SD_BO_11 :=, SD_BO_12 :=, SD_BO_13 :=, SD_BO_14 :=, SD_BO_15 :=, SD_I_00 :=, SD_I_01 :=, SD_DI_00 :=, DINTMODE :=, DP_DP_ID := 2, TIMEOUT := T#1s, LADDR := "Local~Interfaccia_PROFINET_2~F-PEMS01-CORE", ERROR => "Emergency_DB".xSendError, SUBS_ON =>, RET_DPRD =>, RET_DPWR =>, DIAG =>)
   END_RUNG
   // the same network as SCL:
   "Send_Core"(SD_BO_00 := "ESTOP1_DB".Q,   // SENDDP
               SD_BO_01 := "ESTOP1_DB".Q_DELAY,
               SD_BO_02 := "ESTOP2_DB".Q,
               SD_BO_03 := "ESTOP2_DB".Q_DELAY,
               SD_BO_04 := "ESTOP3_DB".Q,
               SD_BO_05 := "ESTOP3_DB".Q_DELAY,
               SD_BO_06 := "Reminder".x1,
               SD_BO_10 := "Emergency stop from PCS1 (PE)",
               DP_DP_ID := 2,
               TIMEOUT := T#1s,
               LADDR := "Local~Interfaccia_PROFINET_2~F-PEMS01-CORE",
               ERROR => "Emergency_DB".xSendError);
END_REGION
END_FUNCTION_BLOCK

FUNCTION "SM1_Logic" : Void   // FC60, LAD
TITLE = State Machine Logic
{ S7_Optimized_Access := 'TRUE' }
VERSION : 0.1
// stored: AutoNumber false, IsIECCheckEnabled false, SetENOAutomatically false, UDAEnableTagReadback false
   VAR_TEMP
      xStopSubSystem : Bool;
   END_VAR
   VAR_TEMP   // added for the SCL form of the ladder/FBD networks
      _w1 : Bool;
   END_VAR
BEGIN

REGION Network 1: Stop Command Local Mode
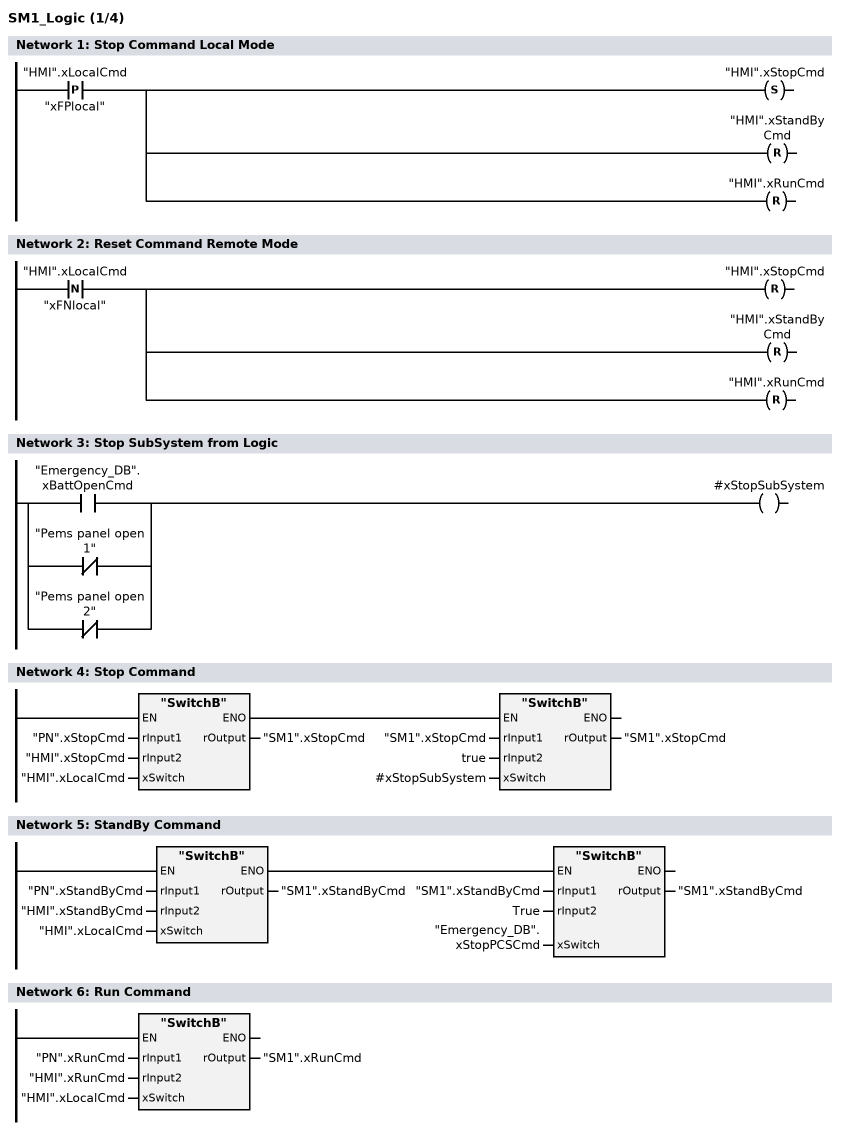
   RUNG wire#powerrail
      P_Contact(operand := "HMI".xLocalCmd, bit := "xFPlocal")
      wire#w1
      S_Coil( "HMI".xStopCmd )
   END_RUNG
   RUNG wire#w1
      R_Coil( "HMI".xStandByCmd )
   END_RUNG
   RUNG wire#w1
      R_Coil( "HMI".xRunCmd )
   END_RUNG
   // the same network as SCL:
   #_w1 := "HMI".xLocalCmd AND NOT "xFPlocal";   // rising edge of "HMI".xLocalCmd
   "xFPlocal" := "HMI".xLocalCmd;
   IF #_w1 THEN
       "HMI".xStopCmd := TRUE;
       "HMI".xStandByCmd := FALSE;
       "HMI".xRunCmd := FALSE;
   END_IF;
END_REGION

REGION Network 2: Reset Command Remote Mode
   RUNG wire#powerrail
      N_Contact(operand := "HMI".xLocalCmd, bit := "xFNlocal")
      wire#w1
      R_Coil( "HMI".xStopCmd )
   END_RUNG
   RUNG wire#w1
      R_Coil( "HMI".xStandByCmd )
   END_RUNG
   RUNG wire#w1
      R_Coil( "HMI".xRunCmd )
   END_RUNG
   // the same network as SCL:
   #_w1 := NOT "HMI".xLocalCmd AND "xFNlocal";   // falling edge of "HMI".xLocalCmd
   "xFNlocal" := "HMI".xLocalCmd;
   IF #_w1 THEN
       "HMI".xStopCmd := FALSE;
       "HMI".xStandByCmd := FALSE;
       "HMI".xRunCmd := FALSE;
   END_IF;
END_REGION

REGION Network 3: Stop SubSystem from Logic
   RUNG wire#powerrail
      Contact( "Emergency_DB".xBattOpenCmd )
      wire#w1
      Coil( #xStopSubSystem )
   END_RUNG
   RUNG wire#powerrail
      I_Contact( "Pems panel open 1" )
   END_RUNG wire#w1
   RUNG wire#powerrail
      I_Contact( "Pems panel open 2" )
   END_RUNG wire#w1
   // the same network as SCL:
   #xStopSubSystem := "Emergency_DB".xBattOpenCmd OR NOT "Pems panel open 1" OR NOT "Pems panel open 2";
END_REGION

REGION Network 4: Stop Command
   RUNG wire#powerrail
      "SwitchB"(rInput1 := "PN".xStopCmd, rInput2 := "HMI".xStopCmd, xSwitch := "HMI".xLocalCmd, rOutput => "SM1".xStopCmd)
      "SwitchB"(rInput1 := "SM1".xStopCmd, rInput2 := true, xSwitch := #xStopSubSystem, rOutput => "SM1".xStopCmd)
   END_RUNG
   // the same network as SCL:
   "SwitchB"(rInput1 := "PN".xStopCmd,
             rInput2 := "HMI".xStopCmd,
             xSwitch := "HMI".xLocalCmd,
             rOutput => "SM1".xStopCmd,
             ENO => #_w1);
   IF #_w1 THEN
       "SwitchB"(rInput1 := "SM1".xStopCmd, rInput2 := true, xSwitch := #xStopSubSystem, rOutput => "SM1".xStopCmd);
   END_IF;
END_REGION

REGION Network 5: StandBy Command
   RUNG wire#powerrail
      "SwitchB"(rInput1 := "PN".xStandByCmd, rInput2 := "HMI".xStandByCmd, xSwitch := "HMI".xLocalCmd, rOutput => "SM1".xStandByCmd)
      "SwitchB"(rInput1 := "SM1".xStandByCmd, rInput2 := True, xSwitch := "Emergency_DB".xStopPCSCmd, rOutput => "SM1".xStandByCmd)
   END_RUNG
   // the same network as SCL:
   "SwitchB"(rInput1 := "PN".xStandByCmd,
             rInput2 := "HMI".xStandByCmd,
             xSwitch := "HMI".xLocalCmd,
             rOutput => "SM1".xStandByCmd,
             ENO => #_w1);
   IF #_w1 THEN
       "SwitchB"(rInput1 := "SM1".xStandByCmd,
                 rInput2 := True,
                 xSwitch := "Emergency_DB".xStopPCSCmd,
                 rOutput => "SM1".xStandByCmd);
   END_IF;
END_REGION

REGION Network 6: Run Command
   RUNG wire#powerrail
      "SwitchB"(rInput1 := "PN".xRunCmd, rInput2 := "HMI".xRunCmd, xSwitch := "HMI".xLocalCmd, rOutput => "SM1".xRunCmd)
   END_RUNG
   // the same network as SCL:
   "SwitchB"(rInput1 := "PN".xRunCmd,
             rInput2 := "HMI".xRunCmd,
             xSwitch := "HMI".xLocalCmd,
             rOutput => "SM1".xRunCmd);
END_REGION

REGION Network 7: Local - Stop - StandBy - Run Status -> to HMI status
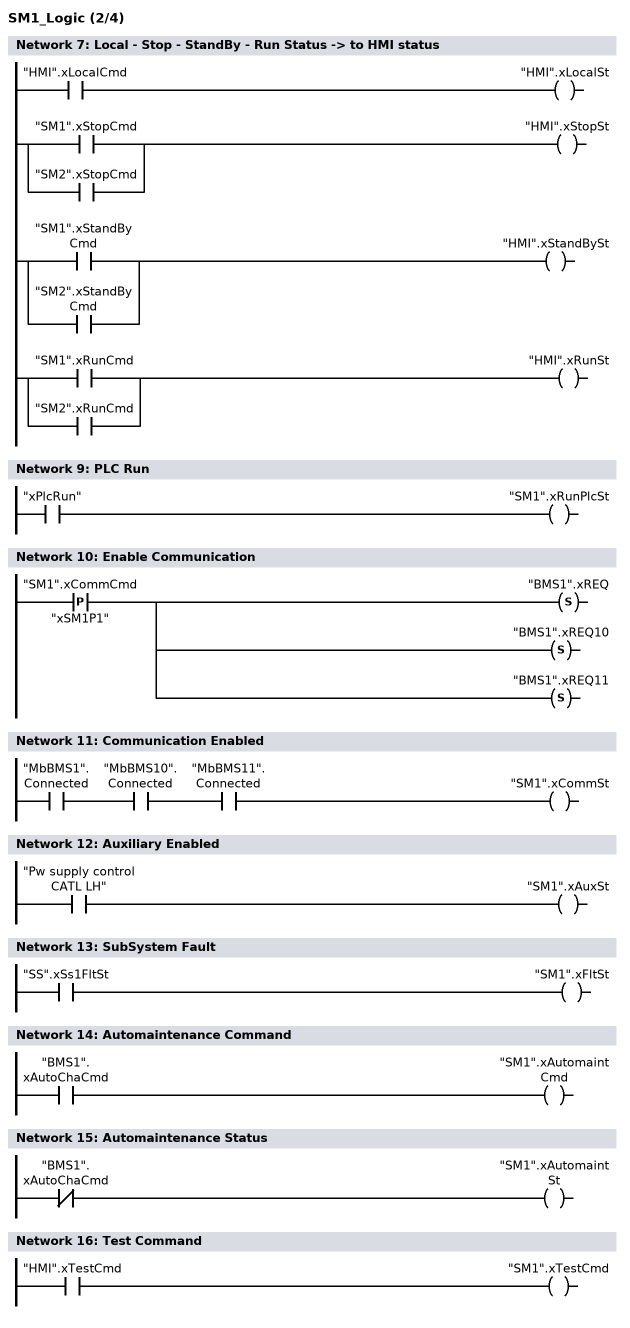
   RUNG wire#powerrail
      Contact( "HMI".xLocalCmd )
      Coil( "HMI".xLocalSt )
   END_RUNG
   RUNG wire#powerrail
      Contact( "SM1".xStopCmd )
      wire#w1
      Coil( "HMI".xStopSt )
   END_RUNG
   RUNG wire#powerrail
      Contact( "SM2".xStopCmd )
   END_RUNG wire#w1
   RUNG wire#powerrail
      Contact( "SM1".xStandByCmd )
      wire#w2
      Coil( "HMI".xStandBySt )
   END_RUNG
   RUNG wire#powerrail
      Contact( "SM2".xStandByCmd )
   END_RUNG wire#w2
   RUNG wire#powerrail
      Contact( "SM1".xRunCmd )
      wire#w3
      Coil( "HMI".xRunSt )
   END_RUNG
   RUNG wire#powerrail
      Contact( "SM2".xRunCmd )
   END_RUNG wire#w3
   // the same network as SCL:
   "HMI".xLocalSt := "HMI".xLocalCmd;
   "HMI".xStopSt := "SM1".xStopCmd OR "SM2".xStopCmd;
   "HMI".xStandBySt := "SM1".xStandByCmd OR "SM2".xStandByCmd;
   "HMI".xRunSt := "SM1".xRunCmd OR "SM2".xRunCmd;
END_REGION

REGION Network 9: PLC Run
   RUNG wire#powerrail
      Contact( "xPlcRun" )
      Coil( "SM1".xRunPlcSt )
   END_RUNG
   // the same network as SCL:
   "SM1".xRunPlcSt := "xPlcRun";
END_REGION

REGION Network 10: Enable Communication
   RUNG wire#powerrail
      P_Contact(operand := "SM1".xCommCmd, bit := "xSM1P1")
      wire#w1
      S_Coil( "BMS1".xREQ )
   END_RUNG
   RUNG wire#w1
      S_Coil( "BMS1".xREQ10 )
   END_RUNG
   RUNG wire#w1
      S_Coil( "BMS1".xREQ11 )
   END_RUNG
   // the same network as SCL:
   #_w1 := "SM1".xCommCmd AND NOT "xSM1P1";   // rising edge of "SM1".xCommCmd
   "xSM1P1" := "SM1".xCommCmd;
   IF #_w1 THEN
       "BMS1".xREQ := TRUE;
       "BMS1".xREQ10 := TRUE;
       "BMS1".xREQ11 := TRUE;
   END_IF;
END_REGION

REGION Network 11: Communication Enabled
   RUNG wire#powerrail
      Contact( "MbBMS1".Connected )
      Contact( "MbBMS10".Connected )
      Contact( "MbBMS11".Connected )
      Coil( "SM1".xCommSt )
   END_RUNG
   // the same network as SCL:
   "SM1".xCommSt := "MbBMS1".Connected AND "MbBMS10".Connected AND "MbBMS11".Connected;
END_REGION

REGION Network 12: Auxiliary Enabled
   RUNG wire#powerrail
      Contact( "Pw supply control CATL LH" )
      Coil( "SM1".xAuxSt )
   END_RUNG
   // the same network as SCL:
   "SM1".xAuxSt := "Pw supply control CATL LH";
END_REGION

REGION Network 13: SubSystem Fault
   RUNG wire#powerrail
      Contact( "SS".xSs1FltSt )
      Coil( "SM1".xFltSt )
   END_RUNG
   // the same network as SCL:
   "SM1".xFltSt := "SS".xSs1FltSt;
END_REGION

REGION Network 14: Automaintenance Command
   RUNG wire#powerrail
      Contact( "BMS1".xAutoChaCmd )
      Coil( "SM1".xAutomaintCmd )
   END_RUNG
   // the same network as SCL:
   "SM1".xAutomaintCmd := "BMS1".xAutoChaCmd;
END_REGION

REGION Network 15: Automaintenance Status
   RUNG wire#powerrail
      I_Contact( "BMS1".xAutoChaCmd )
      Coil( "SM1".xAutomaintSt )
   END_RUNG
   // the same network as SCL:
   "SM1".xAutomaintSt := NOT "BMS1".xAutoChaCmd;
END_REGION

REGION Network 16: Test Command
   RUNG wire#powerrail
      Contact( "HMI".xTestCmd )
      Coil( "SM1".xTestCmd )
   END_RUNG
   // the same network as SCL:
   "SM1".xTestCmd := "HMI".xTestCmd;
END_REGION

REGION Network 17: Ready condition on the Power Island - to check
   // - primo contatto era "MV ok" from PN 
   // -gli altri sono i DC breaker close dei PE
   // -e un bypass icoming UPS line from grid
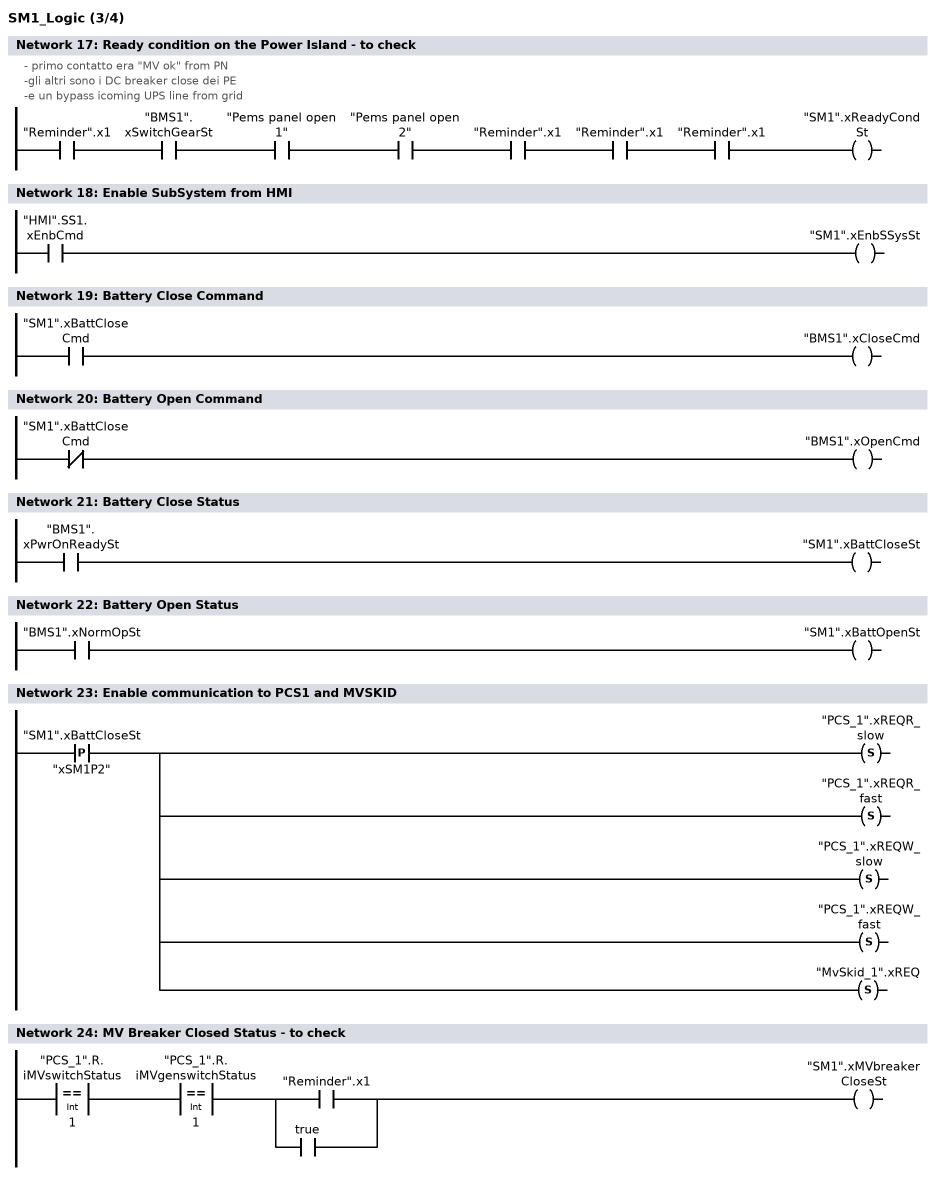
   RUNG wire#powerrail
      Contact( "Reminder".x1 )
      Contact( "BMS1".xSwitchGearSt )
      Contact( "Pems panel open 1" )
      Contact( "Pems panel open 2" )
      Contact( "Reminder".x1 )
      Contact( "Reminder".x1 )
      Contact( "Reminder".x1 )
      Coil( "SM1".xReadyCondSt )
   END_RUNG
   // the same network as SCL:
   "SM1".xReadyCondSt := "Reminder".x1 AND "BMS1".xSwitchGearSt AND "Pems panel open 1" AND "Pems panel open 2" AND "Reminder".x1 AND "Reminder".x1 AND "Reminder".x1;
END_REGION

REGION Network 18: Enable SubSystem from HMI
   RUNG wire#powerrail
      Contact( "HMI".SS1.xEnbCmd )
      Coil( "SM1".xEnbSSysSt )
   END_RUNG
   // the same network as SCL:
   "SM1".xEnbSSysSt := "HMI".SS1.xEnbCmd;
END_REGION

REGION Network 19: Battery Close Command
   RUNG wire#powerrail
      Contact( "SM1".xBattCloseCmd )
      Coil( "BMS1".xCloseCmd )
   END_RUNG
   // the same network as SCL:
   "BMS1".xCloseCmd := "SM1".xBattCloseCmd;
END_REGION

REGION Network 20: Battery Open Command
   RUNG wire#powerrail
      I_Contact( "SM1".xBattCloseCmd )
      Coil( "BMS1".xOpenCmd )
   END_RUNG
   // the same network as SCL:
   "BMS1".xOpenCmd := NOT "SM1".xBattCloseCmd;
END_REGION

REGION Network 21: Battery Close Status
   RUNG wire#powerrail
      Contact( "BMS1".xPwrOnReadySt )
      Coil( "SM1".xBattCloseSt )
   END_RUNG
   // the same network as SCL:
   "SM1".xBattCloseSt := "BMS1".xPwrOnReadySt;
END_REGION

REGION Network 22: Battery Open Status
   RUNG wire#powerrail
      Contact( "BMS1".xNormOpSt )
      Coil( "SM1".xBattOpenSt )
   END_RUNG
   // the same network as SCL:
   "SM1".xBattOpenSt := "BMS1".xNormOpSt;
END_REGION

REGION Network 23: Enable communication to PCS1 and MVSKID
   RUNG wire#powerrail
      P_Contact(operand := "SM1".xBattCloseSt, bit := "xSM1P2")
      wire#w1
      S_Coil( "PCS_1".xREQR_slow )
   END_RUNG
   RUNG wire#w1
      S_Coil( "PCS_1".xREQR_fast )
   END_RUNG
   RUNG wire#w1
      S_Coil( "PCS_1".xREQW_slow )
   END_RUNG
   RUNG wire#w1
      S_Coil( "PCS_1".xREQW_fast )
   END_RUNG
   RUNG wire#w1
      S_Coil( "MvSkid_1".xREQ )
   END_RUNG
   // the same network as SCL:
   #_w1 := "SM1".xBattCloseSt AND NOT "xSM1P2";   // rising edge of "SM1".xBattCloseSt
   "xSM1P2" := "SM1".xBattCloseSt;
   IF #_w1 THEN
       "PCS_1".xREQR_slow := TRUE;
       "PCS_1".xREQR_fast := TRUE;
       "PCS_1".xREQW_slow := TRUE;
       "PCS_1".xREQW_fast := TRUE;
       "MvSkid_1".xREQ := TRUE;
   END_IF;
END_REGION

REGION Network 24: MV Breaker Closed Status - to check
   RUNG wire#powerrail
      { S7_Templates := "SrcType := Int" } EQ_Contact(in1 := "PCS_1".R.iMVswitchStatus, in2 := 1)
      { S7_Templates := "SrcType := Int" } EQ_Contact(in1 := "PCS_1".R.iMVgenswitchStatus, in2 := 1)
      wire#w1
      Contact( "Reminder".x1 )
      wire#w2
      Coil( "SM1".xMVbreakerCloseSt )
   END_RUNG
   RUNG wire#w1
      Contact( true )
   END_RUNG wire#w2
   // the same network as SCL:
   "SM1".xMVbreakerCloseSt := ("PCS_1".R.iMVswitchStatus = 1) AND ("PCS_1".R.iMVgenswitchStatus = 1) AND ("Reminder".x1 OR true);
END_REGION

REGION Network 25: MV Breaker Open Status
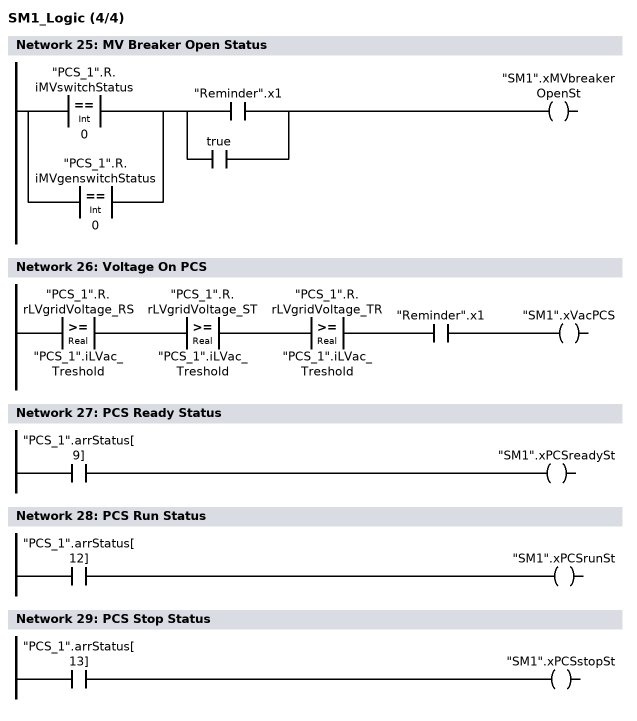
   RUNG wire#powerrail
      { S7_Templates := "SrcType := Int" } EQ_Contact(in1 := "PCS_1".R.iMVswitchStatus, in2 := 0)
      wire#w1
      Contact( "Reminder".x1 )
      wire#w2
      Coil( "SM1".xMVbreakerOpenSt )
   END_RUNG
   RUNG wire#powerrail
      { S7_Templates := "SrcType := Int" } EQ_Contact(in1 := "PCS_1".R.iMVgenswitchStatus, in2 := 0)
   END_RUNG wire#w1
   RUNG wire#w1
      Contact( true )
   END_RUNG wire#w2
   // the same network as SCL:
   "SM1".xMVbreakerOpenSt := (("PCS_1".R.iMVswitchStatus = 0) OR ("PCS_1".R.iMVgenswitchStatus = 0)) AND ("Reminder".x1 OR true);
END_REGION

REGION Network 26: Voltage On PCS
   RUNG wire#powerrail
      { S7_Templates := "SrcType := Real" } GE_Contact(in1 := "PCS_1".R.rLVgridVoltage_RS, in2 := "PCS_1".iLVac_Treshold)
      { S7_Templates := "SrcType := Real" } GE_Contact(in1 := "PCS_1".R.rLVgridVoltage_ST, in2 := "PCS_1".iLVac_Treshold)
      { S7_Templates := "SrcType := Real" } GE_Contact(in1 := "PCS_1".R.rLVgridVoltage_TR, in2 := "PCS_1".iLVac_Treshold)
      Contact( "Reminder".x1 )
      Coil( "SM1".xVacPCS )
   END_RUNG
   // the same network as SCL:
   "SM1".xVacPCS := ("PCS_1".R.rLVgridVoltage_RS >= "PCS_1".iLVac_Treshold) AND ("PCS_1".R.rLVgridVoltage_ST >= "PCS_1".iLVac_Treshold) AND ("PCS_1".R.rLVgridVoltage_TR >= "PCS_1".iLVac_Treshold) AND "Reminder".x1;
END_REGION

REGION Network 27: PCS Ready Status
   RUNG wire#powerrail
      Contact( "PCS_1".arrStatus[9] )
      Coil( "SM1".xPCSreadySt )
   END_RUNG
   // the same network as SCL:
   "SM1".xPCSreadySt := "PCS_1".arrStatus[9];
END_REGION

REGION Network 28: PCS Run Status
   RUNG wire#powerrail
      Contact( "PCS_1".arrStatus[12] )
      Coil( "SM1".xPCSrunSt )
   END_RUNG
   // the same network as SCL:
   "SM1".xPCSrunSt := "PCS_1".arrStatus[12];
END_REGION

REGION Network 29: PCS Stop Status
   RUNG wire#powerrail
      Contact( "PCS_1".arrStatus[13] )
      Coil( "SM1".xPCSstopSt )
   END_RUNG
   // the same network as SCL:
   "SM1".xPCSstopSt := "PCS_1".arrStatus[13];
END_REGION
END_FUNCTION

FUNCTION "SwitchB" : Void
{ S7_Optimized_Access := 'TRUE' }
VERSION : 0.1
   VAR_INPUT 
      rInput1 : Bool;
      rInput2 : Bool;
      xSwitch : Bool;
   END_VAR

   VAR_OUTPUT 
      rOutput : Bool;
   END_VAR

   VAR_TEMP 
      rOutTemp : Bool;
   END_VAR


BEGIN
	IF #xSwitch THEN
	    #rOutTemp := #rInput2;
	ELSE
	    #rOutTemp := #rInput1;
	END_IF;
	
	#rOutput := #rOutTemp;
END_FUNCTION

FUNCTION_BLOCK "State_Machine1"   // FB61, GRAPH
VERSION : 0.1
// stored: AcknowledgeErrorsRequired true, AutoNumber false, GraphVersion 6.0, InitialValuesAcquisition false, IsIECCheckEnabled false, LanguageInNetworks LAD, LockOperatingMode false, PermanentILProcessingInMANMode false, SetENOAutomatically false, SkipSteps false, UDAEnableTagReadback false, WithAlarmHandling true
   // inherited from GRAPH_BASE
   VAR
      OFF_SQ_BASE : Bool;
   END_VAR
   VAR_INPUT
      OFF_SQ { ExternalAccessible := 'False'; ExternalVisible := 'False'; ExternalWritable := 'False'} : Bool := false;   // Disattiva catena / Turn sequence off
      INIT_SQ { ExternalAccessible := 'False'; ExternalVisible := 'False'; ExternalWritable := 'False'} : Bool := false;   // Imposta catena nello stato iniziale / Set sequence to initial state
      ACK_EF { ExternalAccessible := 'False'; ExternalVisible := 'False'; ExternalWritable := 'False'} : Bool := false;   // Conferma tutti gli errori e le anomalie / Acknowledge all errors and faults
      S_PREV { ExternalAccessible := 'False'; ExternalVisible := 'False'; ExternalWritable := 'False'} : Bool := false;   // Emetti il passo precedente nel parametro S_NO / Output previous step in parameter S_NO
      S_NEXT { ExternalAccessible := 'False'; ExternalVisible := 'False'; ExternalWritable := 'False'} : Bool := false;   // Visualizza passo successivo nel parametro S_NO / Indicate next step in parameter S_NO
      SW_AUTO { ExternalAccessible := 'False'; ExternalVisible := 'False'; ExternalWritable := 'False'} : Bool := false;   // Imposta funzionamento automatico / Automatic mode
      SW_TAP { ExternalAccessible := 'False'; ExternalVisible := 'False'; ExternalWritable := 'False'} : Bool := false;   // Semiautomatico/Avanza con transizione / Semiautomatic/switch with transition
      SW_TOP { ExternalAccessible := 'False'; ExternalVisible := 'False'; ExternalWritable := 'False'} : Bool := false;   // Semiautomatico/Ignora transizione / Semiautomatic/ignore transition
      SW_MAN { ExternalAccessible := 'False'; ExternalVisible := 'False'; ExternalWritable := 'False'} : Bool := false;   // Funzionamento manuale / Manual mode
      S_SEL { ExternalAccessible := 'False'; ExternalVisible := 'False'; ExternalWritable := 'False'} : Int := 0;   // Seleziona passo da visualizzare in S_NO / Select step to be output to S_NO
      S_ON { ExternalAccessible := 'False'; ExternalVisible := 'False'; ExternalWritable := 'False'} : Bool := false;   // Attiva passo visualizzato nel parametro S_NO / Activate step indicated in S_NO
      S_OFF { ExternalAccessible := 'False'; ExternalVisible := 'False'; ExternalWritable := 'False'} : Bool := false;   // Disattiva passo visualizzato nel parametro S_NO / Deactivate step indicated S_NO
      T_PUSH { ExternalAccessible := 'False'; ExternalVisible := 'False'; ExternalWritable := 'False'} : Bool := false;   // Abilita commutazione per la transizione nel funzionamento semiautomatico / Enable transition to switch in semi automatic mode
   END_VAR
   VAR_OUTPUT
      S_NO { ExternalAccessible := 'False'; ExternalVisible := 'False'; ExternalWritable := 'False'} : Int := 0;   // Numero del passo / Step number
      S_MORE { ExternalAccessible := 'False'; ExternalVisible := 'False'; ExternalWritable := 'False'} : Bool := false;   // Sono presenti altri passi e possono essere visualizzati in S_NO. / More steps are available and can be shown in S_NO
      S_ACTIVE { ExternalAccessible := 'False'; ExternalVisible := 'False'; ExternalWritable := 'False'} : Bool := false;   // Il passo visualizzato nel parametro S_NO è attivo / Step indicated in S_NO is active
      ERR_FLT { ExternalAccessible := 'False'; ExternalVisible := 'False'; ExternalWritable := 'False'} : Bool := false;   // Errore cumulativo interlock o supervisione / Interlock or supervision group error
      AUTO_ON { ExternalAccessible := 'False'; ExternalVisible := 'False'; ExternalWritable := 'False'} : Bool := false;   // Funzionamento automatico attivo / Automatic mode is active
      TAP_ON { ExternalAccessible := 'False'; ExternalVisible := 'False'; ExternalWritable := 'False'} : Bool := false;   // Funzionamento semiautomatico/Passo con transizione attivo / Semiautomatic mode/step with transition enabled
      TOP_ON { ExternalAccessible := 'False'; ExternalVisible := 'False'; ExternalWritable := 'False'} : Bool := false;   // Semiautomatico/Ignora transizione attivo / Semiautomatic mode/ignore transition enabled
      MAN_ON { ExternalAccessible := 'False'; ExternalVisible := 'False'; ExternalWritable := 'False'} : Bool := false;   // Funzionamento manuale attivo / Manual mode is active
   END_VAR
BEGIN
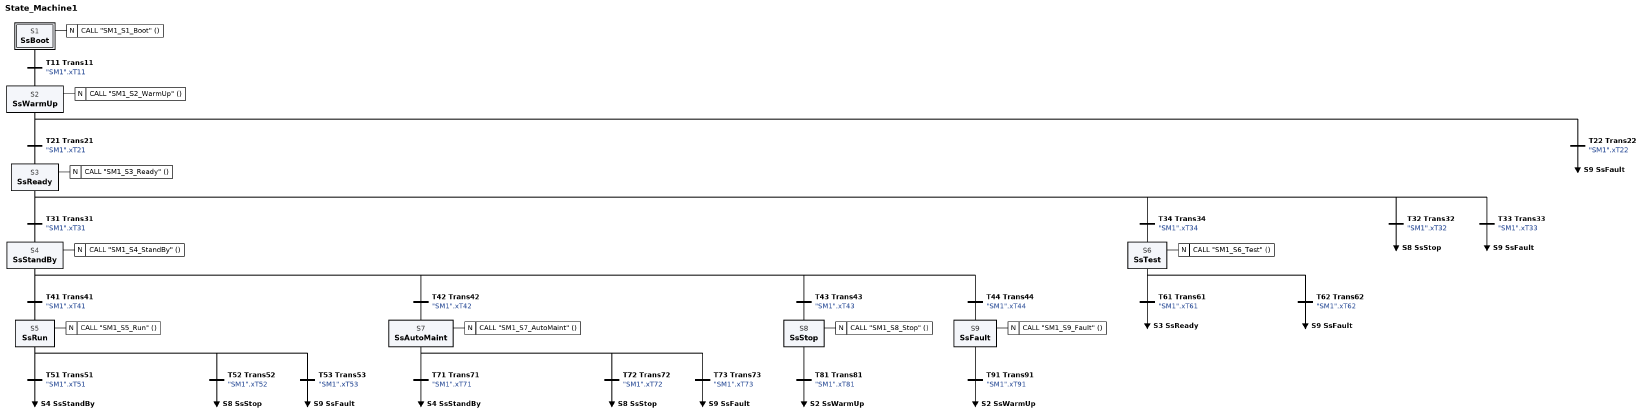
   // sequencer 1: State Machine Battery
   INITIAL_STEP SsBoot:   // S1, max time T#10S, warning time T#7S
              N    CALL "SM1_S1_Boot" ()
   END_STEP
   TRANSITION Trans11 FROM SsBoot TO SsWarmUp   // T11
      := "SM1".xT11;
   END_TRANSITION
   STEP SsWarmUp:   // S2, max time T#10S, warning time T#7S
              N    CALL "SM1_S2_WarmUp" ()
   END_STEP
   TRANSITION Trans21 FROM SsWarmUp TO SsReady   // T21
      := "SM1".xT21;
   END_TRANSITION
   TRANSITION Trans22 FROM SsWarmUp TO SsFault   // T22, jump
      := "SM1".xT22;
   END_TRANSITION
   STEP SsReady:   // S3, max time T#10S, warning time T#7S
              N    CALL "SM1_S3_Ready" ()
   END_STEP
   TRANSITION Trans31 FROM SsReady TO SsStandBy   // T31
      := "SM1".xT31;
   END_TRANSITION
   TRANSITION Trans34 FROM SsReady TO SsTest   // T34
      := "SM1".xT34;
   END_TRANSITION
   TRANSITION Trans32 FROM SsReady TO SsStop   // T32, jump
      := "SM1".xT32;
   END_TRANSITION
   TRANSITION Trans33 FROM SsReady TO SsFault   // T33, jump
      := "SM1".xT33;
   END_TRANSITION
   STEP SsStandBy:   // S4, max time T#10S, warning time T#7S
              N    CALL "SM1_S4_StandBy" ()
   END_STEP
   TRANSITION Trans41 FROM SsStandBy TO SsRun   // T41
      := "SM1".xT41;
   END_TRANSITION
   TRANSITION Trans42 FROM SsStandBy TO SsAutoMaint   // T42
      := "SM1".xT42;
   END_TRANSITION
   TRANSITION Trans43 FROM SsStandBy TO SsStop   // T43
      := "SM1".xT43;
   END_TRANSITION
   TRANSITION Trans44 FROM SsStandBy TO SsFault   // T44
      := "SM1".xT44;
   END_TRANSITION
   STEP SsRun:   // S5, max time T#10S, warning time T#7S
              N    CALL "SM1_S5_Run" ()
   END_STEP
   TRANSITION Trans51 FROM SsRun TO SsStandBy   // T51, jump
      := "SM1".xT51;
   END_TRANSITION
   TRANSITION Trans52 FROM SsRun TO SsStop   // T52, jump
      := "SM1".xT52;
   END_TRANSITION
   TRANSITION Trans53 FROM SsRun TO SsFault   // T53, jump
      := "SM1".xT53;
   END_TRANSITION
   STEP SsTest:   // S6, max time T#10S, warning time T#7S
              N    CALL "SM1_S6_Test" ()
   END_STEP
   TRANSITION Trans61 FROM SsTest TO SsReady   // T61, jump
      := "SM1".xT61;
   END_TRANSITION
   TRANSITION Trans62 FROM SsTest TO SsFault   // T62, jump
      := "SM1".xT62;
   END_TRANSITION
   STEP SsAutoMaint:   // S7, max time T#10S, warning time T#7S
              N    CALL "SM1_S7_AutoMaint" ()
   END_STEP
   TRANSITION Trans71 FROM SsAutoMaint TO SsStandBy   // T71, jump
      := "SM1".xT71;
   END_TRANSITION
   TRANSITION Trans72 FROM SsAutoMaint TO SsStop   // T72, jump
      := "SM1".xT72;
   END_TRANSITION
   TRANSITION Trans73 FROM SsAutoMaint TO SsFault   // T73, jump
      := "SM1".xT73;
   END_TRANSITION
   STEP SsStop:   // S8, max time T#10S, warning time T#7S
              N    CALL "SM1_S8_Stop" ()
   END_STEP
   TRANSITION Trans81 FROM SsStop TO SsWarmUp   // T81, jump
      := "SM1".xT81;
   END_TRANSITION
   STEP SsFault:   // S9, max time T#10S, warning time T#7S
              N    CALL "SM1_S9_Fault" ()
   END_STEP
   TRANSITION Trans91 FROM SsFault TO SsWarmUp   // T91, jump
      := "SM1".xT91;
   END_TRANSITION
END_FUNCTION_BLOCK

FUNCTION "SM2_Logic" : Void   // FC50, LAD
TITLE = State Machine Logic
{ S7_Optimized_Access := 'TRUE' }
VERSION : 0.1
// stored: AutoNumber true, IsIECCheckEnabled false, SetENOAutomatically false, UDAEnableTagReadback false
   VAR_TEMP
      xStopSubSystem : Bool;
   END_VAR
   VAR_TEMP   // added for the SCL form of the ladder/FBD networks
      _w1 : Bool;
   END_VAR
BEGIN

REGION Network 1: Stop Command Local Mode
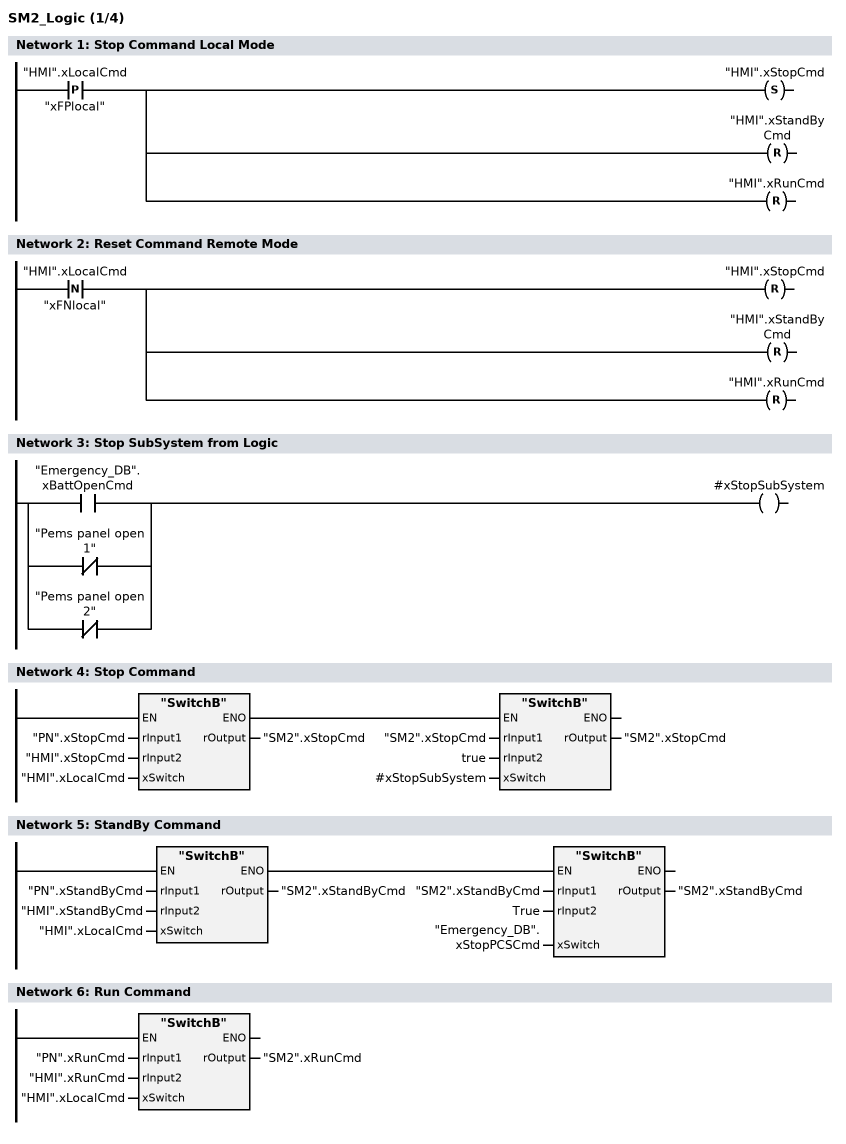
   RUNG wire#powerrail
      P_Contact(operand := "HMI".xLocalCmd, bit := "xFPlocal")
      wire#w1
      S_Coil( "HMI".xStopCmd )
   END_RUNG
   RUNG wire#w1
      R_Coil( "HMI".xStandByCmd )
   END_RUNG
   RUNG wire#w1
      R_Coil( "HMI".xRunCmd )
   END_RUNG
   // the same network as SCL:
   #_w1 := "HMI".xLocalCmd AND NOT "xFPlocal";   // rising edge of "HMI".xLocalCmd
   "xFPlocal" := "HMI".xLocalCmd;
   IF #_w1 THEN
       "HMI".xStopCmd := TRUE;
       "HMI".xStandByCmd := FALSE;
       "HMI".xRunCmd := FALSE;
   END_IF;
END_REGION

REGION Network 2: Reset Command Remote Mode
   RUNG wire#powerrail
      N_Contact(operand := "HMI".xLocalCmd, bit := "xFNlocal")
      wire#w1
      R_Coil( "HMI".xStopCmd )
   END_RUNG
   RUNG wire#w1
      R_Coil( "HMI".xStandByCmd )
   END_RUNG
   RUNG wire#w1
      R_Coil( "HMI".xRunCmd )
   END_RUNG
   // the same network as SCL:
   #_w1 := NOT "HMI".xLocalCmd AND "xFNlocal";   // falling edge of "HMI".xLocalCmd
   "xFNlocal" := "HMI".xLocalCmd;
   IF #_w1 THEN
       "HMI".xStopCmd := FALSE;
       "HMI".xStandByCmd := FALSE;
       "HMI".xRunCmd := FALSE;
   END_IF;
END_REGION

REGION Network 3: Stop SubSystem from Logic
   RUNG wire#powerrail
      Contact( "Emergency_DB".xBattOpenCmd )
      wire#w1
      Coil( #xStopSubSystem )
   END_RUNG
   RUNG wire#powerrail
      I_Contact( "Pems panel open 1" )
   END_RUNG wire#w1
   RUNG wire#powerrail
      I_Contact( "Pems panel open 2" )
   END_RUNG wire#w1
   // the same network as SCL:
   #xStopSubSystem := "Emergency_DB".xBattOpenCmd OR NOT "Pems panel open 1" OR NOT "Pems panel open 2";
END_REGION

REGION Network 4: Stop Command
   RUNG wire#powerrail
      "SwitchB"(rInput1 := "PN".xStopCmd, rInput2 := "HMI".xStopCmd, xSwitch := "HMI".xLocalCmd, rOutput => "SM2".xStopCmd)
      "SwitchB"(rInput1 := "SM2".xStopCmd, rInput2 := true, xSwitch := #xStopSubSystem, rOutput => "SM2".xStopCmd)
   END_RUNG
   // the same network as SCL:
   "SwitchB"(rInput1 := "PN".xStopCmd,
             rInput2 := "HMI".xStopCmd,
             xSwitch := "HMI".xLocalCmd,
             rOutput => "SM2".xStopCmd,
             ENO => #_w1);
   IF #_w1 THEN
       "SwitchB"(rInput1 := "SM2".xStopCmd, rInput2 := true, xSwitch := #xStopSubSystem, rOutput => "SM2".xStopCmd);
   END_IF;
END_REGION

REGION Network 5: StandBy Command
   RUNG wire#powerrail
      "SwitchB"(rInput1 := "PN".xStandByCmd, rInput2 := "HMI".xStandByCmd, xSwitch := "HMI".xLocalCmd, rOutput => "SM2".xStandByCmd)
      "SwitchB"(rInput1 := "SM2".xStandByCmd, rInput2 := True, xSwitch := "Emergency_DB".xStopPCSCmd, rOutput => "SM2".xStandByCmd)
   END_RUNG
   // the same network as SCL:
   "SwitchB"(rInput1 := "PN".xStandByCmd,
             rInput2 := "HMI".xStandByCmd,
             xSwitch := "HMI".xLocalCmd,
             rOutput => "SM2".xStandByCmd,
             ENO => #_w1);
   IF #_w1 THEN
       "SwitchB"(rInput1 := "SM2".xStandByCmd,
                 rInput2 := True,
                 xSwitch := "Emergency_DB".xStopPCSCmd,
                 rOutput => "SM2".xStandByCmd);
   END_IF;
END_REGION

REGION Network 6: Run Command
   RUNG wire#powerrail
      "SwitchB"(rInput1 := "PN".xRunCmd, rInput2 := "HMI".xRunCmd, xSwitch := "HMI".xLocalCmd, rOutput => "SM2".xRunCmd)
   END_RUNG
   // the same network as SCL:
   "SwitchB"(rInput1 := "PN".xRunCmd,
             rInput2 := "HMI".xRunCmd,
             xSwitch := "HMI".xLocalCmd,
             rOutput => "SM2".xRunCmd);
END_REGION

REGION Network 7: Local - Stop - StandBy - Run Status -> to HMI status
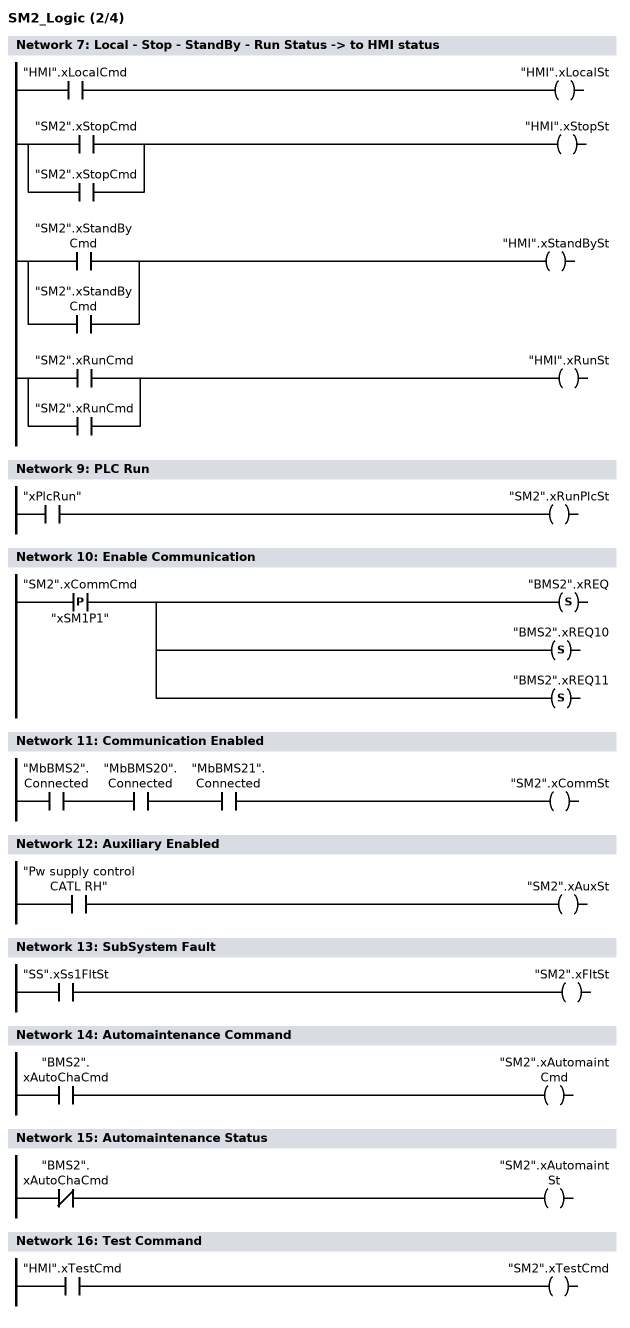
   RUNG wire#powerrail
      Contact( "HMI".xLocalCmd )
      Coil( "HMI".xLocalSt )
   END_RUNG
   RUNG wire#powerrail
      Contact( "SM2".xStopCmd )
      wire#w1
      Coil( "HMI".xStopSt )
   END_RUNG
   RUNG wire#powerrail
      Contact( "SM2".xStopCmd )
   END_RUNG wire#w1
   RUNG wire#powerrail
      Contact( "SM2".xStandByCmd )
      wire#w2
      Coil( "HMI".xStandBySt )
   END_RUNG
   RUNG wire#powerrail
      Contact( "SM2".xStandByCmd )
   END_RUNG wire#w2
   RUNG wire#powerrail
      Contact( "SM2".xRunCmd )
      wire#w3
      Coil( "HMI".xRunSt )
   END_RUNG
   RUNG wire#powerrail
      Contact( "SM2".xRunCmd )
   END_RUNG wire#w3
   // the same network as SCL:
   "HMI".xLocalSt := "HMI".xLocalCmd;
   "HMI".xStopSt := "SM2".xStopCmd OR "SM2".xStopCmd;
   "HMI".xStandBySt := "SM2".xStandByCmd OR "SM2".xStandByCmd;
   "HMI".xRunSt := "SM2".xRunCmd OR "SM2".xRunCmd;
END_REGION

REGION Network 9: PLC Run
   RUNG wire#powerrail
      Contact( "xPlcRun" )
      Coil( "SM2".xRunPlcSt )
   END_RUNG
   // the same network as SCL:
   "SM2".xRunPlcSt := "xPlcRun";
END_REGION

REGION Network 10: Enable Communication
   RUNG wire#powerrail
      P_Contact(operand := "SM2".xCommCmd, bit := "xSM1P1")
      wire#w1
      S_Coil( "BMS2".xREQ )
   END_RUNG
   RUNG wire#w1
      S_Coil( "BMS2".xREQ10 )
   END_RUNG
   RUNG wire#w1
      S_Coil( "BMS2".xREQ11 )
   END_RUNG
   // the same network as SCL:
   #_w1 := "SM2".xCommCmd AND NOT "xSM1P1";   // rising edge of "SM2".xCommCmd
   "xSM1P1" := "SM2".xCommCmd;
   IF #_w1 THEN
       "BMS2".xREQ := TRUE;
       "BMS2".xREQ10 := TRUE;
       "BMS2".xREQ11 := TRUE;
   END_IF;
END_REGION

REGION Network 11: Communication Enabled
   RUNG wire#powerrail
      Contact( "MbBMS2".Connected )
      Contact( "MbBMS20".Connected )
      Contact( "MbBMS21".Connected )
      Coil( "SM2".xCommSt )
   END_RUNG
   // the same network as SCL:
   "SM2".xCommSt := "MbBMS2".Connected AND "MbBMS20".Connected AND "MbBMS21".Connected;
END_REGION

REGION Network 12: Auxiliary Enabled
   RUNG wire#powerrail
      Contact( "Pw supply control CATL RH" )
      Coil( "SM2".xAuxSt )
   END_RUNG
   // the same network as SCL:
   "SM2".xAuxSt := "Pw supply control CATL RH";
END_REGION

REGION Network 13: SubSystem Fault
   RUNG wire#powerrail
      Contact( "SS".xSs1FltSt )
      Coil( "SM2".xFltSt )
   END_RUNG
   // the same network as SCL:
   "SM2".xFltSt := "SS".xSs1FltSt;
END_REGION

REGION Network 14: Automaintenance Command
   RUNG wire#powerrail
      Contact( "BMS2".xAutoChaCmd )
      Coil( "SM2".xAutomaintCmd )
   END_RUNG
   // the same network as SCL:
   "SM2".xAutomaintCmd := "BMS2".xAutoChaCmd;
END_REGION

REGION Network 15: Automaintenance Status
   RUNG wire#powerrail
      I_Contact( "BMS2".xAutoChaCmd )
      Coil( "SM2".xAutomaintSt )
   END_RUNG
   // the same network as SCL:
   "SM2".xAutomaintSt := NOT "BMS2".xAutoChaCmd;
END_REGION

REGION Network 16: Test Command
   RUNG wire#powerrail
      Contact( "HMI".xTestCmd )
      Coil( "SM2".xTestCmd )
   END_RUNG
   // the same network as SCL:
   "SM2".xTestCmd := "HMI".xTestCmd;
END_REGION

REGION Network 17: Ready condition on the Power Island - to check
   // - primo contatto era "MV ok" from PN 
   // -gli altri sono i DC breaker close dei PE
   // -e un bypass icoming UPS line from grid
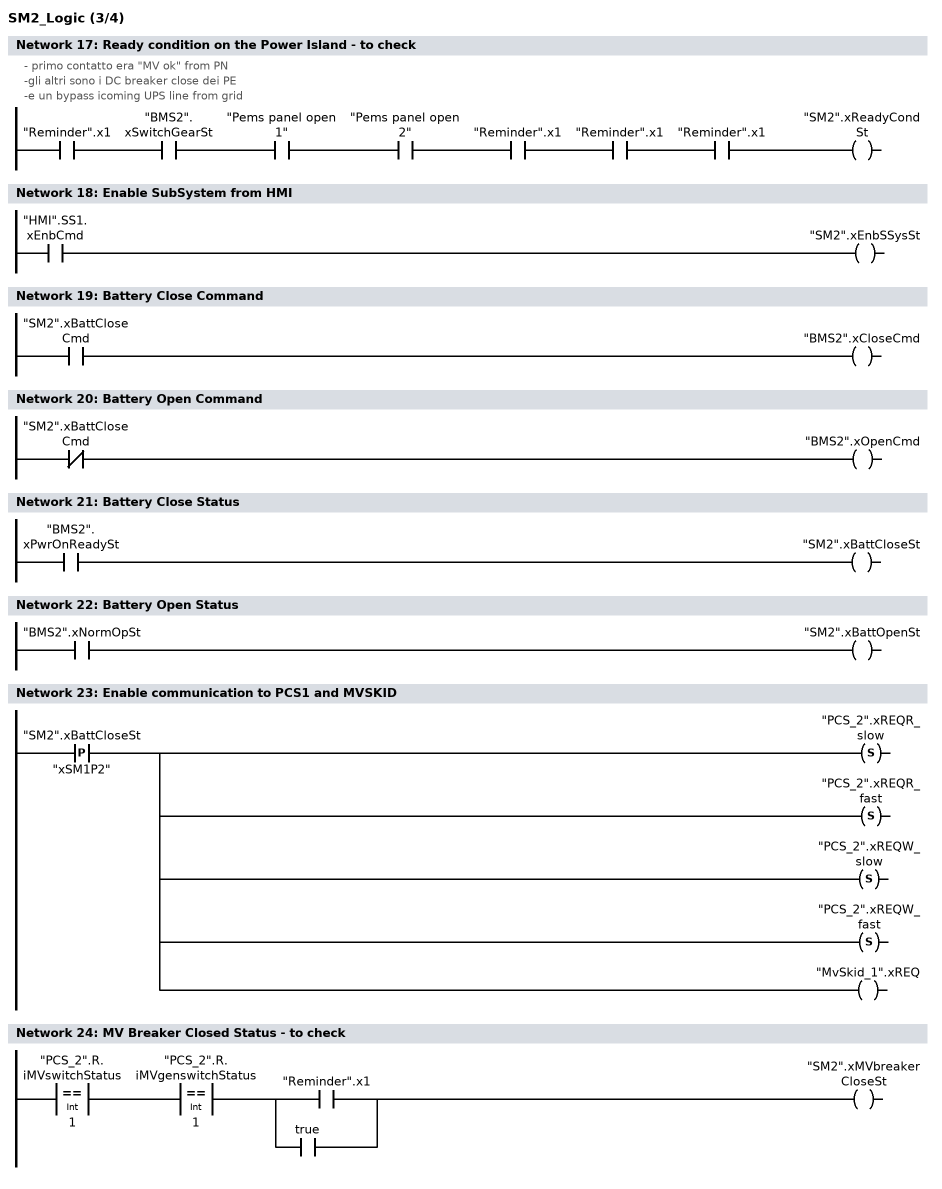
   RUNG wire#powerrail
      Contact( "Reminder".x1 )
      Contact( "BMS2".xSwitchGearSt )
      Contact( "Pems panel open 1" )
      Contact( "Pems panel open 2" )
      Contact( "Reminder".x1 )
      Contact( "Reminder".x1 )
      Contact( "Reminder".x1 )
      Coil( "SM2".xReadyCondSt )
   END_RUNG
   // the same network as SCL:
   "SM2".xReadyCondSt := "Reminder".x1 AND "BMS2".xSwitchGearSt AND "Pems panel open 1" AND "Pems panel open 2" AND "Reminder".x1 AND "Reminder".x1 AND "Reminder".x1;
END_REGION

REGION Network 18: Enable SubSystem from HMI
   RUNG wire#powerrail
      Contact( "HMI".SS1.xEnbCmd )
      Coil( "SM2".xEnbSSysSt )
   END_RUNG
   // the same network as SCL:
   "SM2".xEnbSSysSt := "HMI".SS1.xEnbCmd;
END_REGION

REGION Network 19: Battery Close Command
   RUNG wire#powerrail
      Contact( "SM2".xBattCloseCmd )
      Coil( "BMS2".xCloseCmd )
   END_RUNG
   // the same network as SCL:
   "BMS2".xCloseCmd := "SM2".xBattCloseCmd;
END_REGION

REGION Network 20: Battery Open Command
   RUNG wire#powerrail
      I_Contact( "SM2".xBattCloseCmd )
      Coil( "BMS2".xOpenCmd )
   END_RUNG
   // the same network as SCL:
   "BMS2".xOpenCmd := NOT "SM2".xBattCloseCmd;
END_REGION

REGION Network 21: Battery Close Status
   RUNG wire#powerrail
      Contact( "BMS2".xPwrOnReadySt )
      Coil( "SM2".xBattCloseSt )
   END_RUNG
   // the same network as SCL:
   "SM2".xBattCloseSt := "BMS2".xPwrOnReadySt;
END_REGION

REGION Network 22: Battery Open Status
   RUNG wire#powerrail
      Contact( "BMS2".xNormOpSt )
      Coil( "SM2".xBattOpenSt )
   END_RUNG
   // the same network as SCL:
   "SM2".xBattOpenSt := "BMS2".xNormOpSt;
END_REGION

REGION Network 23: Enable communication to PCS1 and MVSKID
   RUNG wire#powerrail
      P_Contact(operand := "SM2".xBattCloseSt, bit := "xSM1P2")
      wire#w1
      S_Coil( "PCS_2".xREQR_slow )
   END_RUNG
   RUNG wire#w1
      S_Coil( "PCS_2".xREQR_fast )
   END_RUNG
   RUNG wire#w1
      S_Coil( "PCS_2".xREQW_slow )
   END_RUNG
   RUNG wire#w1
      S_Coil( "PCS_2".xREQW_fast )
   END_RUNG
   RUNG wire#w1
      Coil( "MvSkid_1".xREQ )
   END_RUNG
   // the same network as SCL:
   #_w1 := "SM2".xBattCloseSt AND NOT "xSM1P2";   // rising edge of "SM2".xBattCloseSt
   "xSM1P2" := "SM2".xBattCloseSt;
   IF #_w1 THEN
       "PCS_2".xREQR_slow := TRUE;
       "PCS_2".xREQR_fast := TRUE;
       "PCS_2".xREQW_slow := TRUE;
       "PCS_2".xREQW_fast := TRUE;
   END_IF;
   "MvSkid_1".xREQ := #_w1;
END_REGION

REGION Network 24: MV Breaker Closed Status - to check
   RUNG wire#powerrail
      { S7_Templates := "SrcType := Int" } EQ_Contact(in1 := "PCS_2".R.iMVswitchStatus, in2 := 1)
      { S7_Templates := "SrcType := Int" } EQ_Contact(in1 := "PCS_2".R.iMVgenswitchStatus, in2 := 1)
      wire#w1
      Contact( "Reminder".x1 )
      wire#w2
      Coil( "SM2".xMVbreakerCloseSt )
   END_RUNG
   RUNG wire#w1
      Contact( true )
   END_RUNG wire#w2
   // the same network as SCL:
   "SM2".xMVbreakerCloseSt := ("PCS_2".R.iMVswitchStatus = 1) AND ("PCS_2".R.iMVgenswitchStatus = 1) AND ("Reminder".x1 OR true);
END_REGION

REGION Network 25: MV Breaker Open Status
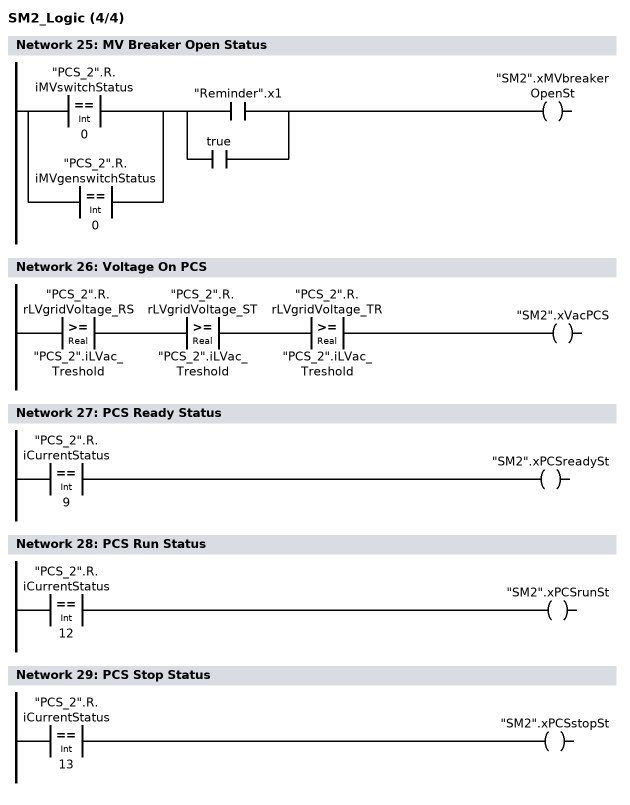
   RUNG wire#powerrail
      { S7_Templates := "SrcType := Int" } EQ_Contact(in1 := "PCS_2".R.iMVswitchStatus, in2 := 0)
      wire#w1
      Contact( "Reminder".x1 )
      wire#w2
      Coil( "SM2".xMVbreakerOpenSt )
   END_RUNG
   RUNG wire#powerrail
      { S7_Templates := "SrcType := Int" } EQ_Contact(in1 := "PCS_2".R.iMVgenswitchStatus, in2 := 0)
   END_RUNG wire#w1
   RUNG wire#w1
      Contact( true )
   END_RUNG wire#w2
   // the same network as SCL:
   "SM2".xMVbreakerOpenSt := (("PCS_2".R.iMVswitchStatus = 0) OR ("PCS_2".R.iMVgenswitchStatus = 0)) AND ("Reminder".x1 OR true);
END_REGION

REGION Network 26: Voltage On PCS
   RUNG wire#powerrail
      { S7_Templates := "SrcType := Real" } GE_Contact(in1 := "PCS_2".R.rLVgridVoltage_RS, in2 := "PCS_2".iLVac_Treshold)
      { S7_Templates := "SrcType := Real" } GE_Contact(in1 := "PCS_2".R.rLVgridVoltage_ST, in2 := "PCS_2".iLVac_Treshold)
      { S7_Templates := "SrcType := Real" } GE_Contact(in1 := "PCS_2".R.rLVgridVoltage_TR, in2 := "PCS_2".iLVac_Treshold)
      Coil( "SM2".xVacPCS )
   END_RUNG
   // the same network as SCL:
   "SM2".xVacPCS := ("PCS_2".R.rLVgridVoltage_RS >= "PCS_2".iLVac_Treshold) AND ("PCS_2".R.rLVgridVoltage_ST >= "PCS_2".iLVac_Treshold) AND ("PCS_2".R.rLVgridVoltage_TR >= "PCS_2".iLVac_Treshold);
END_REGION

REGION Network 27: PCS Ready Status
   RUNG wire#powerrail
      { S7_Templates := "SrcType := Int" } EQ_Contact(in1 := "PCS_2".R.iCurrentStatus, in2 := 9)
      Coil( "SM2".xPCSreadySt )
   END_RUNG
   // the same network as SCL:
   "SM2".xPCSreadySt := "PCS_2".R.iCurrentStatus = 9;
END_REGION

REGION Network 28: PCS Run Status
   RUNG wire#powerrail
      { S7_Templates := "SrcType := Int" } EQ_Contact(in1 := "PCS_2".R.iCurrentStatus, in2 := 12)
      Coil( "SM2".xPCSrunSt )
   END_RUNG
   // the same network as SCL:
   "SM2".xPCSrunSt := "PCS_2".R.iCurrentStatus = 12;
END_REGION

REGION Network 29: PCS Stop Status
   RUNG wire#powerrail
      { S7_Templates := "SrcType := Int" } EQ_Contact(in1 := "PCS_2".R.iCurrentStatus, in2 := 13)
      Coil( "SM2".xPCSstopSt )
   END_RUNG
   // the same network as SCL:
   "SM2".xPCSstopSt := "PCS_2".R.iCurrentStatus = 13;
END_REGION
END_FUNCTION

